LIN {X 0,Y 491.694,Z 547.992,A -85,B 0,C 180,E1 -6473.64,E2 -6473.64} C_VEL
LIN {X 0,Y 488.846,Z 539.593,A -85,B 0,C 180,E1 -6473.888,E2 -6473.888} C_VEL
LIN {X 0,Y 488.957,Z 539.577,A -85,B 0,C 180,E1 -6477.529,E2 -6477.529} C_VEL
LIN {X 0,Y 488.958,Z 539.578,A -85,B 0,C 180,E1 -6480,E2 -6480} C_VEL
LIN {X 0,Y 488.952,Z 539.582,A -85,B 0,C 180,E1 -6482.471,E2 -6482.471} C_VEL
LIN {X 0,Y 488.863,Z 539.586,A -85,B 0,C 180,E1 -6485.776,E2 -6485.776} C_VEL
LIN {X 0,Y 488.808,Z 539.594,A -85,B 0,C 180,E1 -6488.267,E2 -6488.267} C_VEL
LIN {X 0,Y 488.82,Z 539.592,A -85,B 0,C 180,E1 -6491.612,E2 -6491.612} C_VEL
LIN {X 0,Y 488.753,Z 539.602,A -85,B 0,C 180,E1 -6495.001,E2 -6495.001} C_VEL
LIN {X 0,Y 488.744,Z 539.606,A -85,B 0,C 180,E1 -6498.443,E2 -6498.443} C_VEL
LIN {X 0,Y 488.697,Z 539.611,A -85,B 0,C 180,E1 -6501.071,E2 -6501.071} C_VEL
LIN {X 0,Y 488.683,Z 539.609,A -85,B 0,C 180,E1 -6503.746,E2 -6503.746} C_VEL
LIN {X 0,Y 488.789,Z 539.601,A -85,B 0,C 180,E1 -6506.946,E2 -6506.946} C_VEL
LIN {X 0,Y 488.71,Z 539.608,A -85,B 0,C 180,E1 -6510.366,E2 -6510.366} C_VEL
LIN {X 0,Y 488.728,Z 539.604,A -85,B 0,C 180,E1 -6513.485,E2 -6513.485} C_VEL
LIN {X 0,Y 488.682,Z 539.612,A -85,B 0,C 180,E1 -6516.357,E2 -6516.357} C_VEL
LIN {X 0,Y 488.742,Z 539.604,A -85,B 0,C 180,E1 -6519.251,E2 -6519.251} C_VEL
LIN {X 0,Y 488.728,Z 539.609,A -85,B 0,C 180,E1 -6522.522,E2 -6522.522} C_VEL
LIN {X 0,Y 488.706,Z 539.611,A -85,B 0,C 180,E1 -6525.2,E2 -6525.2} C_VEL
LIN {X 0,Y 488.73,Z 539.605,A -85,B 0,C 180,E1 -6527.48,E2 -6527.48} C_VEL
LIN {X 0,Y 488.744,Z 539.607,A -85,B 0,C 180,E1 -6530.752,E2 -6530.752} C_VEL
LIN {X 0,Y 488.683,Z 539.612,A -85,B 0,C 180,E1 -6533.87,E2 -6533.87} C_VEL
LIN {X 0,Y 488.737,Z 539.61,A -85,B 0,C 180,E1 -6536.878,E2 -6536.878} C_VEL
LIN {X 0,Y 488.796,Z 539.749,A -85,B 0,C 180,E1 -6540.411,E2 -6540.411} C_VEL
LIN {X 0,Y 491.958,Z 554.443,A -85,B 0,C 180,E1 -6542.55,E2 -6542.55} C_VEL
LIN {X 0,Y 491.604,Z 568.227,A -85,B 0,C 180,E1 -6544.347,E2 -6544.347} C_VEL
LIN {X 0,Y 490.777,Z 592.773,A -85,B 0,C 180,E1 -6547.478,E2 -6547.478} C_VEL
LIN {X 0,Y 490.123,Z 615.461,A -85,B 0,C 180,E1 -6550.309,E2 -6550.309} C_VEL
LIN {X 0,Y 489.503,Z 641.425,A -85,B 0,C 180,E1 -6553.507,E2 -6553.507} C_VEL
LIN {X 0,Y 489.465,Z 643.124,A -85,B 0,C 180,E1 -6553.715,E2 -6553.715} C_VEL
LIN {X 0,Y 491.552,Z 663.555,A -85,B 0,C 180,E1 -6554.102,E2 -6554.102} C_VEL
LIN {X 0,Y 490.879,Z 754.427,A -85,B 0,C 180,E1 -6555.491,E2 -6555.491} C_VEL
LIN {X 0,Y 490.504,Z 768.429,A -85,B 0,C 180,E1 -6555.877,E2 -6555.877} C_VEL
LIN {X 0,Y 490.138,Z 781.627,A -85,B 0,C 180,E1 -6556.421,E2 -6556.421} C_VEL
LIN {X 0,Y 489.854,Z 793.54,A -85,B 0,C 180,E1 -6557.047,E2 -6557.047} C_VEL
LIN {X 0,Y 489.551,Z 804.345,A -85,B 0,C 180,E1 -6557.776,E2 -6557.776} C_VEL
LIN {X 0,Y 489.111,Z 815.314,A -85,B 0,C 180,E1 -6558.711,E2 -6558.711} C_VEL
LIN {X 0,Y 488.793,Z 824.213,A -85,B 0,C 180,E1 -6559.647,E2 -6559.647} C_VEL
LIN {X 0,Y 488.538,Z 832.373,A -85,B 0,C 180,E1 -6560.687,E2 -6560.687} C_VEL
LIN {X 0,Y 488.332,Z 840.353,A -85,B 0,C 180,E1 -6561.934,E2 -6561.934} C_VEL
LIN {X 0,Y 488.188,Z 845.733,A -85,B 0,C 180,E1 -6562.972,E2 -6562.972} C_VEL
LIN {X 0,Y 488.147,Z 850.985,A -85,B 0,C 180,E1 -6564.217,E2 -6564.217} C_VEL
LIN {X 0,Y 488.028,Z 855.04,A -85,B 0,C 180,E1 -6565.458,E2 -6565.458} C_VEL
LIN {X 0,Y 488.064,Z 858.028,A -85,B 0,C 180,E1 -6566.699,E2 -6566.699} C_VEL
LIN {X 0,Y 488.013,Z 859.461,A -85,B 0,C 180,E1 -6567.525,E2 -6567.525} C_VEL
LIN {X 0,Y 487.957,Z 861.087,A -85,B 0,C 180,E1 -6569.175,E2 -6569.175} C_VEL
LIN {X 0,Y 487.966,Z 861.309,A -85,B 0,C 180,E1 -6570.001,E2 -6570.001} C_VEL
LIN {X 0,Y 487.964,Z 860.468,A -85,B 0,C 180,E1 -6571.651,E2 -6571.651} C_VEL
LIN {X 0,Y 488.002,Z 859.457,A -85,B 0,C 180,E1 -6572.477,E2 -6572.477} C_VEL
LIN {X 0,Y 488.033,Z 858.023,A -85,B 0,C 180,E1 -6573.303,E2 -6573.303} C_VEL
LIN {X 0,Y 488.022,Z 855.034,A -85,B 0,C 180,E1 -6574.544,E2 -6574.544} C_VEL
LIN {X 0,Y 488.147,Z 849.944,A -85,B 0,C 180,E1 -6576.05,E2 -6576.05} C_VEL
LIN {X 0,Y 488.207,Z 843.696,A -85,B 0,C 180,E1 -6577.445,E2 -6577.445} C_VEL
LIN {X 0,Y 488.433,Z 836.567,A -85,B 0,C 180,E1 -6578.69,E2 -6578.69} C_VEL
LIN {X 0,Y 488.667,Z 827.667,A -85,B 0,C 180,E1 -6579.939,E2 -6579.939} C_VEL
LIN {X 0,Y 488.999,Z 818.502,A -85,B 0,C 180,E1 -6580.979,E2 -6580.979} C_VEL
LIN {X 0,Y 489.377,Z 808.262,A -85,B 0,C 180,E1 -6581.914,E2 -6581.914} C_VEL
LIN {X 0,Y 489.69,Z 797.091,A -85,B 0,C 180,E1 -6582.738,E2 -6582.738} C_VEL
LIN {X 0,Y 490.104,Z 784.736,A -85,B 0,C 180,E1 -6583.476,E2 -6583.476} C_VEL
LIN {X 0,Y 490.522,Z 771.929,A -85,B 0,C 180,E1 -6584.045,E2 -6584.045} C_VEL
LIN {X 0,Y 490.842,Z 759.389,A -85,B 0,C 180,E1 -6584.432,E2 -6584.432} C_VEL
LIN {X 0,Y 491.06,Z 742.038,A -85,B 0,C 180,E1 -6584.743,E2 -6584.743} C_VEL
LIN {X 0,Y 491.516,Z 663.042,A -85,B 0,C 180,E1 -6585.933,E2 -6585.933} C_VEL
LIN {X 0,Y 489.357,Z 645.546,A -85,B 0,C 180,E1 -6586.287,E2 -6586.287} C_VEL
LIN {X 0,Y 489.969,Z 622.617,A -85,B 0,C 180,E1 -6589.481,E2 -6589.481} C_VEL
LIN {X 0,Y 490.634,Z 601.006,A -85,B 0,C 180,E1 -6592.531,E2 -6592.531} C_VEL
LIN {X 0,Y 491.434,Z 579.535,A -85,B 0,C 180,E1 -6595.603,E2 -6595.603} C_VEL
LIN {X 0,Y 492.217,Z 559.133,A -85,B 0,C 180,E1 -6598.576,E2 -6598.576} C_VEL
LIN {X 0,Y 492.12,Z 554.913,A -85,B 0,C 180,E1 -6599.212,E2 -6599.212} C_VEL
LIN {X 0,Y 488.728,Z 539.608,A -85,B 0,C 180,E1 -6601.733,E2 -6601.733} C_VEL
LIN {X 0,Y 488.735,Z 539.604,A -85,B 0,C 180,E1 -6604.113,E2 -6604.113} C_VEL
LIN {X 0,Y 488.682,Z 539.616,A -85,B 0,C 180,E1 -6607.159,E2 -6607.159} C_VEL
LIN {X 0,Y 488.72,Z 539.605,A -85,B 0,C 180,E1 -6610.345,E2 -6610.345} C_VEL
LIN {X 0,Y 488.689,Z 539.604,A -85,B 0,C 180,E1 -6613.654,E2 -6613.654} C_VEL
LIN {X 0,Y 488.718,Z 539.604,A -85,B 0,C 180,E1 -6616.349,E2 -6616.349} C_VEL
LIN {X 0,Y 488.734,Z 539.604,A -85,B 0,C 180,E1 -6619.677,E2 -6619.677} C_VEL
LIN {X 0,Y 488.684,Z 539.61,A -85,B 0,C 180,E1 -6622.841,E2 -6622.841} C_VEL
LIN {X 0,Y 488.736,Z 539.603,A -85,B 0,C 180,E1 -6625.887,E2 -6625.887} C_VEL
LIN {X 0,Y 488.693,Z 539.605,A -85,B 0,C 180,E1 -6628.82,E2 -6628.82} C_VEL
LIN {X 0,Y 488.745,Z 539.604,A -85,B 0,C 180,E1 -6631.671,E2 -6631.671} C_VEL
LIN {X 0,Y 488.747,Z 539.595,A -85,B 0,C 180,E1 -6634.444,E2 -6634.444} C_VEL
LIN {X 0,Y 488.723,Z 539.604,A -85,B 0,C 180,E1 -6637.153,E2 -6637.153} C_VEL
LIN {X 0,Y 488.725,Z 539.604,A -85,B 0,C 180,E1 -6639.81,E2 -6639.81} C_VEL
LIN {X 0,Y 488.733,Z 539.592,A -85,B 0,C 180,E1 -6642.423,E2 -6642.423} C_VEL
LIN {X 0,Y 488.764,Z 539.599,A -85,B 0,C 180,E1 -6645,E2 -6645} C_VEL
LIN {X 0,Y 488.805,Z 539.587,A -85,B 0,C 180,E1 -6648.388,E2 -6648.388} C_VEL
LIN {X 0,Y 488.818,Z 539.597,A -85,B 0,C 180,E1 -6651.734,E2 -6651.734} C_VEL
LIN {X 0,Y 488.855,Z 539.587,A -85,B 0,C 180,E1 -6654.224,E2 -6654.224} C_VEL
LIN {X 0,Y 488.961,Z 539.57,A -85,B 0,C 180,E1 -6657.529,E2 -6657.529} C_VEL
LIN {X 0,Y 488.954,Z 539.574,A -85,B 0,C 180,E1 -6660.824,E2 -6660.824} C_VEL
LIN {X 0,Y 488.961,Z 539.572,A -85,B 0,C 180,E1 -6662.471,E2 -6662.471} C_VEL
LIN {X 0,Y 488.855,Z 539.584,A -85,B 0,C 180,E1 -6665.776,E2 -6665.776} C_VEL
LIN {X 0,Y 488.817,Z 539.594,A -85,B 0,C 180,E1 -6668.266,E2 -6668.266} C_VEL
LIN {X 0,Y 488.805,Z 539.594,A -85,B 0,C 180,E1 -6671.613,E2 -6671.613} C_VEL
LIN {X 0,Y 488.762,Z 539.597,A -85,B 0,C 180,E1 -6675,E2 -6675} C_VEL
LIN {X 0,Y 488.755,Z 539.594,A -85,B 0,C 180,E1 -6678.442,E2 -6678.442} C_VEL
LIN {X 0,Y 488.707,Z 539.603,A -85,B 0,C 180,E1 -6681.071,E2 -6681.071} C_VEL
LIN {X 0,Y 488.694,Z 539.612,A -85,B 0,C 180,E1 -6683.746,E2 -6683.746} C_VEL
LIN {X 0,Y 488.792,Z 539.593,A -85,B 0,C 180,E1 -6686.944,E2 -6686.944} C_VEL
LIN {X 0,Y 488.71,Z 539.605,A -85,B 0,C 180,E1 -6690.363,E2 -6690.363} C_VEL
LIN {X 0,Y 488.735,Z 539.604,A -85,B 0,C 180,E1 -6693.484,E2 -6693.484} C_VEL
LIN {X 0,Y 488.683,Z 539.615,A -85,B 0,C 180,E1 -6696.355,E2 -6696.355} C_VEL
LIN {X 0,Y 488.703,Z 539.605,A -85,B 0,C 180,E1 -6699.254,E2 -6699.254} C_VEL
LIN {X 0,Y 488.71,Z 539.607,A -85,B 0,C 180,E1 -6701.6,E2 -6701.6} C_VEL
LIN {X 0,Y 488.703,Z 539.608,A -85,B 0,C 180,E1 -6704.803,E2 -6704.803} C_VEL
LIN {X 0,Y 488.69,Z 539.598,A -85,B 0,C 180,E1 -6707.474,E2 -6707.474} C_VEL
LIN {X 0,Y 488.735,Z 539.604,A -85,B 0,C 180,E1 -6709.677,E2 -6709.677} C_VEL
LIN {X 0,Y 488.682,Z 539.612,A -85,B 0,C 180,E1 -6712.841,E2 -6712.841} C_VEL
LIN {X 0,Y 488.736,Z 539.606,A -85,B 0,C 180,E1 -6715.887,E2 -6715.887} C_VEL
LIN {X 0,Y 488.696,Z 539.616,A -85,B 0,C 180,E1 -6718.82,E2 -6718.82} C_VEL
LIN {X 0,Y 488.788,Z 539.603,A -85,B 0,C 180,E1 -6722.17,E2 -6722.17} C_VEL
LIN {X 0,Y 489.997,Z 545.204,A -85,B 0,C 180,E1 -6723.021,E2 -6723.021} C_VEL
LIN {X 0,Y 490.113,Z 548.909,A -85,B 0,C 180,E1 -6723.557,E2 -6723.557} C_VEL
LIN {X 0,Y 489.104,Z 552.826,A -85,B 0,C 180,E1 -6724.068,E2 -6724.068} C_VEL
LIN {X 0,Y 485.091,Z 563.467,A -85,B 0,C 180,E1 -6725.412,E2 -6725.412} C_VEL
LIN {X 0,Y 484.682,Z 566.068,A -85,B 0,C 180,E1 -6725.772,E2 -6725.772} C_VEL
LIN {X 0,Y 483.859,Z 586.48,A -85,B 0,C 180,E1 -6728.708,E2 -6728.708} C_VEL
LIN {X 0,Y 483.266,Z 606.74,A -85,B 0,C 180,E1 -6731.56,E2 -6731.56} C_VEL
LIN {X 0,Y 482.955,Z 621.519,A -85,B 0,C 180,E1 -6733.543,E2 -6733.543} C_VEL
LIN {X 0,Y 484.937,Z 634.789,A -85,B 0,C 180,E1 -6733.814,E2 -6733.814} C_VEL
LIN {X 0,Y 484.351,Z 730.687,A -85,B 0,C 180,E1 -6735.263,E2 -6735.263} C_VEL
LIN {X 0,Y 484.065,Z 743.533,A -85,B 0,C 180,E1 -6735.603,E2 -6735.603} C_VEL
LIN {X 0,Y 483.672,Z 756.506,A -85,B 0,C 180,E1 -6736.128,E2 -6736.128} C_VEL
LIN {X 0,Y 483.242,Z 769.444,A -85,B 0,C 180,E1 -6736.855,E2 -6736.855} C_VEL
LIN {X 0,Y 482.846,Z 781.021,A -85,B 0,C 180,E1 -6737.709,E2 -6737.709} C_VEL
LIN {X 0,Y 482.346,Z 792.291,A -85,B 0,C 180,E1 -6738.762,E2 -6738.762} C_VEL
LIN {X 0,Y 482.016,Z 800.524,A -85,B 0,C 180,E1 -6739.711,E2 -6739.711} C_VEL
LIN {X 0,Y 481.685,Z 808.123,A -85,B 0,C 180,E1 -6740.764,E2 -6740.764} C_VEL
LIN {X 0,Y 481.365,Z 815.544,A -85,B 0,C 180,E1 -6742.027,E2 -6742.027} C_VEL
LIN {X 0,Y 481.126,Z 821.834,A -85,B 0,C 180,E1 -6743.367,E2 -6743.367} C_VEL
LIN {X 0,Y 481.021,Z 826.219,A -85,B 0,C 180,E1 -6744.55,E2 -6744.55} C_VEL
LIN {X 0,Y 480.943,Z 829.827,A -85,B 0,C 180,E1 -6745.809,E2 -6745.809} C_VEL
LIN {X 0,Y 480.908,Z 831.685,A -85,B 0,C 180,E1 -6746.648,E2 -6746.648} C_VEL
LIN {X 0,Y 480.846,Z 833.109,A -85,B 0,C 180,E1 -6747.486,E2 -6747.486} C_VEL
LIN {X 0,Y 480.823,Z 834.106,A -85,B 0,C 180,E1 -6748.324,E2 -6748.324} C_VEL
LIN {X 0,Y 480.743,Z 834.962,A -85,B 0,C 180,E1 -6749.999,E2 -6749.999} C_VEL
LIN {X 0,Y 480.823,Z 834.192,A -85,B 0,C 180,E1 -6751.674,E2 -6751.674} C_VEL
LIN {X 0,Y 480.908,Z 831.872,A -85,B 0,C 180,E1 -6753.35,E2 -6753.35} C_VEL
LIN {X 0,Y 480.899,Z 829.015,A -85,B 0,C 180,E1 -6754.61,E2 -6754.61} C_VEL
LIN {X 0,Y 481.1,Z 825.127,A -85,B 0,C 180,E1 -6755.868,E2 -6755.868} C_VEL
LIN {X 0,Y 481.191,Z 820.1,A -85,B 0,C 180,E1 -6757.131,E2 -6757.131} C_VEL
LIN {X 0,Y 481.41,Z 813.759,A -85,B 0,C 180,E1 -6758.394,E2 -6758.394} C_VEL
LIN {X 0,Y 481.748,Z 805.871,A -85,B 0,C 180,E1 -6759.657,E2 -6759.657} C_VEL
LIN {X 0,Y 482.07,Z 797.812,A -85,B 0,C 180,E1 -6760.712,E2 -6760.712} C_VEL
LIN {X 0,Y 482.573,Z 787.935,A -85,B 0,C 180,E1 -6761.764,E2 -6761.764} C_VEL
LIN {X 0,Y 482.996,Z 776.744,A -85,B 0,C 180,E1 -6762.721,E2 -6762.721} C_VEL
LIN {X 0,Y 483.377,Z 766.004,A -85,B 0,C 180,E1 -6763.451,E2 -6763.451} C_VEL
LIN {X 0,Y 483.783,Z 753.895,A -85,B 0,C 180,E1 -6764.082,E2 -6764.082} C_VEL
LIN {X 0,Y 484.14,Z 740.567,A -85,B 0,C 180,E1 -6764.581,E2 -6764.581} C_VEL
LIN {X 0,Y 484.367,Z 727.094,A -85,B 0,C 180,E1 -6764.897,E2 -6764.897} C_VEL
LIN {X 0,Y 484.82,Z 635.15,A -85,B 0,C 180,E1 -6766.274,E2 -6766.274} C_VEL
LIN {X 0,Y 482.662,Z 622.172,A -85,B 0,C 180,E1 -6766.566,E2 -6766.566} C_VEL
LIN {X 0,Y 483.144,Z 602.516,A -85,B 0,C 180,E1 -6769.545,E2 -6769.545} C_VEL
LIN {X 0,Y 483.734,Z 584.445,A -85,B 0,C 180,E1 -6772.418,E2 -6772.418} C_VEL
LIN {X 0,Y 484.377,Z 566.321,A -85,B 0,C 180,E1 -6775.341,E2 -6775.341} C_VEL
LIN {X 0,Y 484.651,Z 554.986,A -85,B 0,C 180,E1 -6777.179,E2 -6777.179} C_VEL
LIN {X 0,Y 482.201,Z 542.669,A -85,B 0,C 180,E1 -6779.28,E2 -6779.28} C_VEL
LIN {X 0,Y 481.699,Z 540.486,A -85,B 0,C 180,E1 -6779.685,E2 -6779.685} C_VEL
LIN {X 0,Y 481.671,Z 540.486,A -85,B 0,C 180,E1 -6782.673,E2 -6782.673} C_VEL
LIN {X 0,Y 481.64,Z 540.488,A -85,B 0,C 180,E1 -6785.708,E2 -6785.708} C_VEL
LIN {X 0,Y 481.668,Z 540.488,A -85,B 0,C 180,E1 -6788.858,E2 -6788.858} C_VEL
LIN {X 0,Y 481.658,Z 540.484,A -85,B 0,C 180,E1 -6791.913,E2 -6791.913} C_VEL
LIN {X 0,Y 481.654,Z 540.48,A -85,B 0,C 180,E1 -6794.456,E2 -6794.456} C_VEL
LIN {X 0,Y 481.683,Z 540.483,A -85,B 0,C 180,E1 -6796.845,E2 -6796.845} C_VEL
LIN {X 0,Y 481.687,Z 540.483,A -85,B 0,C 180,E1 -6800.06,E2 -6800.06} C_VEL
LIN {X 0,Y 481.681,Z 540.499,A -85,B 0,C 180,E1 -6802.043,E2 -6802.043} C_VEL
LIN {X 0,Y 484.76,Z 549.63,A -85,B 0,C 180,E1 -6802.296,E2 -6802.296} C_VEL
LIN {X 0,Y 484.229,Z 619.899,A -85,B 0,C 180,E1 -6803.411,E2 -6803.411} C_VEL
LIN {X 0,Y 484.143,Z 632.566,A -85,B 0,C 180,E1 -6803.766,E2 -6803.766} C_VEL
LIN {X 0,Y 484.01,Z 645.447,A -85,B 0,C 180,E1 -6804.301,E2 -6804.301} C_VEL
LIN {X 0,Y 483.712,Z 657.474,A -85,B 0,C 180,E1 -6804.977,E2 -6804.977} C_VEL
LIN {X 0,Y 483.368,Z 668.816,A -85,B 0,C 180,E1 -6805.803,E2 -6805.803} C_VEL
LIN {X 0,Y 483.007,Z 679.79,A -85,B 0,C 180,E1 -6806.807,E2 -6806.807} C_VEL
LIN {X 0,Y 482.626,Z 689.455,A -85,B 0,C 180,E1 -6807.916,E2 -6807.916} C_VEL
LIN {X 0,Y 482.342,Z 697.942,A -85,B 0,C 180,E1 -6809.12,E2 -6809.12} C_VEL
LIN {X 0,Y 482.034,Z 704.631,A -85,B 0,C 180,E1 -6810.283,E2 -6810.283} C_VEL
LIN {X 0,Y 481.791,Z 711.107,A -85,B 0,C 180,E1 -6811.7,E2 -6811.7} C_VEL
LIN {X 0,Y 481.666,Z 715.997,A -85,B 0,C 180,E1 -6813.107,E2 -6813.107} C_VEL
LIN {X 0,Y 481.58,Z 718.529,A -85,B 0,C 180,E1 -6814.036,E2 -6814.036} C_VEL
LIN {X 0,Y 481.487,Z 720.459,A -85,B 0,C 180,E1 -6814.957,E2 -6814.957} C_VEL
LIN {X 0,Y 481.429,Z 721.907,A -85,B 0,C 180,E1 -6815.874,E2 -6815.874} C_VEL
LIN {X 0,Y 481.389,Z 722.929,A -85,B 0,C 180,E1 -6816.888,E2 -6816.888} C_VEL
LIN {X 0,Y 481.405,Z 723.32,A -85,B 0,C 180,E1 -6817.693,E2 -6817.693} C_VEL
LIN {X 0,Y 481.417,Z 723.133,A -85,B 0,C 180,E1 -6819.112,E2 -6819.112} C_VEL
LIN {X 0,Y 481.477,Z 721.986,A -85,B 0,C 180,E1 -6820.383,E2 -6820.383} C_VEL
LIN {X 0,Y 481.598,Z 720.132,A -85,B 0,C 180,E1 -6821.536,E2 -6821.536} C_VEL
LIN {X 0,Y 481.746,Z 716.495,A -85,B 0,C 180,E1 -6823.036,E2 -6823.036} C_VEL
LIN {X 0,Y 481.951,Z 711.888,A -85,B 0,C 180,E1 -6824.4,E2 -6824.4} C_VEL
LIN {X 0,Y 482.242,Z 705.298,A -85,B 0,C 180,E1 -6825.871,E2 -6825.871} C_VEL
LIN {X 0,Y 482.564,Z 697.739,A -85,B 0,C 180,E1 -6827.189,E2 -6827.189} C_VEL
LIN {X 0,Y 482.835,Z 690.295,A -85,B 0,C 180,E1 -6828.242,E2 -6828.242} C_VEL
LIN {X 0,Y 483.213,Z 681.009,A -85,B 0,C 180,E1 -6829.313,E2 -6829.313} C_VEL
LIN {X 0,Y 483.592,Z 670.655,A -85,B 0,C 180,E1 -6830.273,E2 -6830.273} C_VEL
LIN {X 0,Y 483.918,Z 659.298,A -85,B 0,C 180,E1 -6831.115,E2 -6831.115} C_VEL
LIN {X 0,Y 484.181,Z 646.995,A -85,B 0,C 180,E1 -6831.811,E2 -6831.811} C_VEL
LIN {X 0,Y 484.306,Z 633.622,A -85,B 0,C 180,E1 -6832.364,E2 -6832.364} C_VEL
LIN {X 0,Y 484.364,Z 620.986,A -85,B 0,C 180,E1 -6832.706,E2 -6832.706} C_VEL
LIN {X 0,Y 484.864,Z 549.455,A -85,B 0,C 180,E1 -6833.863,E2 -6833.863} C_VEL
LIN {X 0,Y 481.827,Z 540.469,A -85,B 0,C 180,E1 -6834.14,E2 -6834.14} C_VEL
LIN {X 0,Y 481.924,Z 540.453,A -85,B 0,C 180,E1 -6837.492,E2 -6837.492} C_VEL
LIN {X 0,Y 481.929,Z 540.454,A -85,B 0,C 180,E1 -6840,E2 -6840} C_VEL
LIN {X 0,Y 481.919,Z 540.458,A -85,B 0,C 180,E1 -6842.507,E2 -6842.507} C_VEL
LIN {X 0,Y 481.821,Z 540.464,A -85,B 0,C 180,E1 -6845.86,E2 -6845.86} C_VEL
LIN {X 0,Y 481.753,Z 540.474,A -85,B 0,C 180,E1 -6848.388,E2 -6848.388} C_VEL
LIN {X 0,Y 481.784,Z 540.469,A -85,B 0,C 180,E1 -6851.784,E2 -6851.784} C_VEL
LIN {X 0,Y 481.733,Z 540.473,A -85,B 0,C 180,E1 -6855.225,E2 -6855.225} C_VEL
LIN {X 0,Y 481.702,Z 540.485,A -85,B 0,C 180,E1 -6858.722,E2 -6858.722} C_VEL
LIN {X 0,Y 481.637,Z 540.488,A -85,B 0,C 180,E1 -6861.395,E2 -6861.395} C_VEL
LIN {X 0,Y 481.667,Z 540.484,A -85,B 0,C 180,E1 -6864.114,E2 -6864.114} C_VEL
LIN {X 0,Y 481.742,Z 540.476,A -85,B 0,C 180,E1 -6867.141,E2 -6867.141} C_VEL
LIN {X 0,Y 481.679,Z 540.481,A -85,B 0,C 180,E1 -6869.741,E2 -6869.741} C_VEL
LIN {X 0,Y 481.665,Z 540.489,A -85,B 0,C 180,E1 -6872.675,E2 -6872.675} C_VEL
LIN {X 0,Y 481.636,Z 540.487,A -85,B 0,C 180,E1 -6875.71,E2 -6875.71} C_VEL
LIN {X 0,Y 481.713,Z 540.479,A -85,B 0,C 180,E1 -6879.356,E2 -6879.356} C_VEL
LIN {X 0,Y 481.669,Z 540.485,A -85,B 0,C 180,E1 -6882.159,E2 -6882.159} C_VEL
LIN {X 0,Y 481.654,Z 540.49,A -85,B 0,C 180,E1 -6884.458,E2 -6884.458} C_VEL
LIN {X 0,Y 481.684,Z 540.487,A -85,B 0,C 180,E1 -6886.847,E2 -6886.847} C_VEL
LIN {X 0,Y 481.688,Z 540.482,A -85,B 0,C 180,E1 -6890.062,E2 -6890.062} C_VEL
LIN {X 0,Y 481.628,Z 540.494,A -85,B 0,C 180,E1 -6893.255,E2 -6893.255} C_VEL
LIN {X 0,Y 481.706,Z 540.482,A -85,B 0,C 180,E1 -6896.331,E2 -6896.331} C_VEL
LIN {X 0,Y 481.69,Z 540.486,A -85,B 0,C 180,E1 -6899.778,E2 -6899.778} C_VEL
LIN {X 0,Y 481.682,Z 540.506,A -85,B 0,C 180,E1 -6900.14,E2 -6900.14} C_VEL
LIN {X 0,Y 484.991,Z 555.483,A -85,B 0,C 180,E1 -6902.374,E2 -6902.374} C_VEL
LIN {X 0,Y 484.898,Z 563.926,A -85,B 0,C 180,E1 -6903.51,E2 -6903.51} C_VEL
LIN {X 0,Y 484.044,Z 586.865,A -85,B 0,C 180,E1 -6906.502,E2 -6906.502} C_VEL
LIN {X 0,Y 483.295,Z 609.138,A -85,B 0,C 180,E1 -6909.352,E2 -6909.352} C_VEL
LIN {X 0,Y 482.634,Z 633.496,A -85,B 0,C 180,E1 -6912.414,E2 -6912.414} C_VEL
LIN {X 0,Y 482.43,Z 641.831,A -85,B 0,C 180,E1 -6913.454,E2 -6913.454} C_VEL
LIN {X 0,Y 484.679,Z 663.774,A -85,B 0,C 180,E1 -6913.893,E2 -6913.893} C_VEL
LIN {X 0,Y 483.941,Z 753.875,A -85,B 0,C 180,E1 -6915.305,E2 -6915.305} C_VEL
LIN {X 0,Y 483.538,Z 767.693,A -85,B 0,C 180,E1 -6915.696,E2 -6915.696} C_VEL
LIN {X 0,Y 483.233,Z 781.439,A -85,B 0,C 180,E1 -6916.223,E2 -6916.223} C_VEL
LIN {X 0,Y 482.906,Z 793.909,A -85,B 0,C 180,E1 -6916.889,E2 -6916.889} C_VEL
LIN {X 0,Y 482.515,Z 805.432,A -85,B 0,C 180,E1 -6917.694,E2 -6917.694} C_VEL
LIN {X 0,Y 482.09,Z 816.209,A -85,B 0,C 180,E1 -6918.651,E2 -6918.651} C_VEL
LIN {X 0,Y 481.713,Z 825.818,A -85,B 0,C 180,E1 -6919.706,E2 -6919.706} C_VEL
LIN {X 0,Y 481.439,Z 833.672,A -85,B 0,C 180,E1 -6920.76,E2 -6920.76} C_VEL
LIN {X 0,Y 481.23,Z 841.303,A -85,B 0,C 180,E1 -6922.026,E2 -6922.026} C_VEL
LIN {X 0,Y 481.028,Z 848.192,A -85,B 0,C 180,E1 -6923.468,E2 -6923.468} C_VEL
LIN {X 0,Y 481.023,Z 852.248,A -85,B 0,C 180,E1 -6924.551,E2 -6924.551} C_VEL
LIN {X 0,Y 480.97,Z 855.936,A -85,B 0,C 180,E1 -6925.811,E2 -6925.811} C_VEL
LIN {X 0,Y 480.986,Z 857.836,A -85,B 0,C 180,E1 -6926.65,E2 -6926.65} C_VEL
LIN {X 0,Y 480.922,Z 859.268,A -85,B 0,C 180,E1 -6927.488,E2 -6927.488} C_VEL
LIN {X 0,Y 480.897,Z 860.278,A -85,B 0,C 180,E1 -6928.326,E2 -6928.326} C_VEL
LIN {X 0,Y 480.875,Z 860.895,A -85,B 0,C 180,E1 -6929.163,E2 -6929.163} C_VEL
LIN {X 0,Y 480.881,Z 861.116,A -85,B 0,C 180,E1 -6930.001,E2 -6930.001} C_VEL
LIN {X 0,Y 480.891,Z 860.276,A -85,B 0,C 180,E1 -6931.676,E2 -6931.676} C_VEL
LIN {X 0,Y 480.911,Z 859.265,A -85,B 0,C 180,E1 -6932.513,E2 -6932.513} C_VEL
LIN {X 0,Y 480.958,Z 857.831,A -85,B 0,C 180,E1 -6933.351,E2 -6933.351} C_VEL
LIN {X 0,Y 480.931,Z 854.843,A -85,B 0,C 180,E1 -6934.611,E2 -6934.611} C_VEL
LIN {X 0,Y 481.047,Z 850.789,A -85,B 0,C 180,E1 -6935.87,E2 -6935.87} C_VEL
LIN {X 0,Y 481.116,Z 844.521,A -85,B 0,C 180,E1 -6937.344,E2 -6937.344} C_VEL
LIN {X 0,Y 481.329,Z 837.682,A -85,B 0,C 180,E1 -6938.608,E2 -6938.608} C_VEL
LIN {X 0,Y 481.532,Z 830.689,A -85,B 0,C 180,E1 -6939.663,E2 -6939.663} C_VEL
LIN {X 0,Y 481.801,Z 822.23,A -85,B 0,C 180,E1 -6940.719,E2 -6940.719} C_VEL
LIN {X 0,Y 482.209,Z 811.732,A -85,B 0,C 180,E1 -6941.774,E2 -6941.774} C_VEL
LIN {X 0,Y 482.535,Z 801.308,A -85,B 0,C 180,E1 -6942.62,E2 -6942.62} C_VEL
LIN {X 0,Y 482.982,Z 789.785,A -85,B 0,C 180,E1 -6943.357,E2 -6943.357} C_VEL
LIN {X 0,Y 483.485,Z 774.679,A -85,B 0,C 180,E1 -6944.093,E2 -6944.093} C_VEL
LIN {X 0,Y 483.852,Z 761.919,A -85,B 0,C 180,E1 -6944.538,E2 -6944.538} C_VEL
LIN {X 0,Y 484.123,Z 748.987,A -85,B 0,C 180,E1 -6944.825,E2 -6944.825} C_VEL
LIN {X 0,Y 484.641,Z 663.611,A -85,B 0,C 180,E1 -6946.143,E2 -6946.143} C_VEL
LIN {X 0,Y 482.358,Z 644.648,A -85,B 0,C 180,E1 -6946.534,E2 -6946.534} C_VEL
LIN {X 0,Y 483.014,Z 621.8,A -85,B 0,C 180,E1 -6949.773,E2 -6949.773} C_VEL
LIN {X 0,Y 483.71,Z 600.186,A -85,B 0,C 180,E1 -6952.872,E2 -6952.872} C_VEL
LIN {X 0,Y 484.565,Z 578.409,A -85,B 0,C 180,E1 -6956.042,E2 -6956.042} C_VEL
LIN {X 0,Y 485.377,Z 558.339,A -85,B 0,C 180,E1 -6959.017,E2 -6959.017} C_VEL
LIN {X 0,Y 484.249,Z 551.933,A -85,B 0,C 180,E1 -6960.046,E2 -6960.046} C_VEL
LIN {X 0,Y 481.663,Z 540.488,A -85,B 0,C 180,E1 -6962,E2 -6962} C_VEL
LIN {X 0,Y 481.693,Z 540.485,A -85,B 0,C 180,E1 -6964.682,E2 -6964.682} C_VEL
LIN {X 0,Y 481.657,Z 540.484,A -85,B 0,C 180,E1 -6968.007,E2 -6968.007} C_VEL
LIN {X 0,Y 481.658,Z 540.491,A -85,B 0,C 180,E1 -6971.042,E2 -6971.042} C_VEL
LIN {X 0,Y 481.661,Z 540.479,A -85,B 0,C 180,E1 -6974.457,E2 -6974.457} C_VEL
LIN {X 0,Y 481.685,Z 540.485,A -85,B 0,C 180,E1 -6976.846,E2 -6976.846} C_VEL
LIN {X 0,Y 481.678,Z 540.481,A -85,B 0,C 180,E1 -6980.06,E2 -6980.06} C_VEL
LIN {X 0,Y 481.63,Z 540.487,A -85,B 0,C 180,E1 -6983.253,E2 -6983.253} C_VEL
LIN {X 0,Y 481.71,Z 540.477,A -85,B 0,C 180,E1 -6986.33,E2 -6986.33} C_VEL
LIN {X 0,Y 481.651,Z 540.484,A -85,B 0,C 180,E1 -6989.417,E2 -6989.417} C_VEL
LIN {X 0,Y 481.7,Z 540.478,A -85,B 0,C 180,E1 -6992.168,E2 -6992.168} C_VEL
LIN {X 0,Y 481.717,Z 540.474,A -85,B 0,C 180,E1 -6994.97,E2 -6994.97} C_VEL
LIN {X 0,Y 481.649,Z 540.489,A -85,B 0,C 180,E1 -6997.705,E2 -6997.705} C_VEL
LIN {X 0,Y 481.705,Z 540.474,A -85,B 0,C 180,E1 -7000.393,E2 -7000.393} C_VEL
LIN {X 0,Y 481.691,Z 540.472,A -85,B 0,C 180,E1 -7003.034,E2 -7003.034} C_VEL
LIN {X 0,Y 481.694,Z 540.485,A -85,B 0,C 180,E1 -7005.639,E2 -7005.639} C_VEL
LIN {X 0,Y 481.75,Z 540.466,A -85,B 0,C 180,E1 -7008.215,E2 -7008.215} C_VEL
LIN {X 0,Y 481.763,Z 540.473,A -85,B 0,C 180,E1 -7011.612,E2 -7011.612} C_VEL
LIN {X 0,Y 481.816,Z 540.464,A -85,B 0,C 180,E1 -7014.14,E2 -7014.14} C_VEL
LIN {X 0,Y 481.927,Z 540.445,A -85,B 0,C 180,E1 -7017.493,E2 -7017.493} C_VEL
LIN {X 0,Y 481.905,Z 540.452,A -85,B 0,C 180,E1 -7020.836,E2 -7020.836} C_VEL
LIN {X 0,Y 481.928,Z 540.448,A -85,B 0,C 180,E1 -7022.508,E2 -7022.508} C_VEL
LIN {X 0,Y 481.816,Z 540.462,A -85,B 0,C 180,E1 -7025.86,E2 -7025.86} C_VEL
LIN {X 0,Y 481.763,Z 540.472,A -85,B 0,C 180,E1 -7028.388,E2 -7028.388} C_VEL
LIN {X 0,Y 481.75,Z 540.47,A -85,B 0,C 180,E1 -7031.785,E2 -7031.785} C_VEL
LIN {X 0,Y 481.742,Z 540.473,A -85,B 0,C 180,E1 -7035.224,E2 -7035.224} C_VEL
LIN {X 0,Y 481.712,Z 540.469,A -85,B 0,C 180,E1 -7038.722,E2 -7038.722} C_VEL
LIN {X 0,Y 481.646,Z 540.484,A -85,B 0,C 180,E1 -7041.395,E2 -7041.395} C_VEL
LIN {X 0,Y 481.678,Z 540.482,A -85,B 0,C 180,E1 -7044.113,E2 -7044.113} C_VEL
LIN {X 0,Y 481.747,Z 540.471,A -85,B 0,C 180,E1 -7047.139,E2 -7047.139} C_VEL
LIN {X 0,Y 481.679,Z 540.484,A -85,B 0,C 180,E1 -7049.741,E2 -7049.741} C_VEL
LIN {X 0,Y 481.672,Z 540.484,A -85,B 0,C 180,E1 -7052.674,E2 -7052.674} C_VEL
LIN {X 0,Y 481.637,Z 540.486,A -85,B 0,C 180,E1 -7055.71,E2 -7055.71} C_VEL
LIN {X 0,Y 481.672,Z 540.481,A -85,B 0,C 180,E1 -7058.859,E2 -7058.859} C_VEL
LIN {X 0,Y 481.655,Z 540.49,A -85,B 0,C 180,E1 -7061.913,E2 -7061.913} C_VEL
LIN {X 0,Y 481.657,Z 540.489,A -85,B 0,C 180,E1 -7064.458,E2 -7064.458} C_VEL
LIN {X 0,Y 481.648,Z 540.477,A -85,B 0,C 180,E1 -7067.839,E2 -7067.839} C_VEL
LIN {X 0,Y 481.682,Z 540.482,A -85,B 0,C 180,E1 -7070.651,E2 -7070.651} C_VEL
LIN {X 0,Y 481.631,Z 540.488,A -85,B 0,C 180,E1 -7073.376,E2 -7073.376} C_VEL
LIN {X 0,Y 481.713,Z 540.484,A -85,B 0,C 180,E1 -7076.33,E2 -7076.33} C_VEL
LIN {X 0,Y 481.654,Z 540.49,A -85,B 0,C 180,E1 -7079.417,E2 -7079.417} C_VEL
LIN {X 0,Y 481.738,Z 540.673,A -85,B 0,C 180,E1 -7081.963,E2 -7081.963} C_VEL
LIN {X 0,Y 484.878,Z 555.303,A -85,B 0,C 180,E1 -7084.225,E2 -7084.225} C_VEL
LIN {X 0,Y 484.682,Z 566.068,A -85,B 0,C 180,E1 -7085.772,E2 -7085.772} C_VEL
LIN {X 0,Y 483.831,Z 569.916,A -85,B 0,C 180,E1 -7086.294,E2 -7086.294} C_VEL
LIN {X 0,Y 477.705,Z 582.954,A -85,B 0,C 180,E1 -7087.927,E2 -7087.927} C_VEL
LIN {X 0,Y 476.962,Z 586.803,A -85,B 0,C 180,E1 -7088.46,E2 -7088.46} C_VEL
LIN {X 0,Y 476.346,Z 606.679,A -85,B 0,C 180,E1 -7091.282,E2 -7091.282} C_VEL
LIN {X 0,Y 476.055,Z 621.776,A -85,B 0,C 180,E1 -7093.3,E2 -7093.3} C_VEL
LIN {X 0,Y 478.157,Z 636.429,A -85,B 0,C 180,E1 -7093.602,E2 -7093.602} C_VEL
LIN {X 0,Y 477.455,Z 732.033,A -85,B 0,C 180,E1 -7095.072,E2 -7095.072} C_VEL
LIN {X 0,Y 477.154,Z 745.254,A -85,B 0,C 180,E1 -7095.444,E2 -7095.444} C_VEL
LIN {X 0,Y 476.751,Z 757.717,A -85,B 0,C 180,E1 -7095.976,E2 -7095.976} C_VEL
LIN {X 0,Y 476.322,Z 769.933,A -85,B 0,C 180,E1 -7096.681,E2 -7096.681} C_VEL
LIN {X 0,Y 475.926,Z 781.195,A -85,B 0,C 180,E1 -7097.527,E2 -7097.527} C_VEL
LIN {X 0,Y 475.373,Z 792.472,A -85,B 0,C 180,E1 -7098.595,E2 -7098.595} C_VEL
LIN {X 0,Y 475.035,Z 800.708,A -85,B 0,C 180,E1 -7099.558,E2 -7099.558} C_VEL
LIN {X 0,Y 474.658,Z 808.311,A -85,B 0,C 180,E1 -7100.626,E2 -7100.626} C_VEL
LIN {X 0,Y 474.319,Z 815.733,A -85,B 0,C 180,E1 -7101.907,E2 -7101.907} C_VEL
LIN {X 0,Y 474.075,Z 822.332,A -85,B 0,C 180,E1 -7103.343,E2 -7103.343} C_VEL
LIN {X 0,Y 473.971,Z 826.411,A -85,B 0,C 180,E1 -7104.469,E2 -7104.469} C_VEL
LIN {X 0,Y 473.845,Z 830.02,A -85,B 0,C 180,E1 -7105.746,E2 -7105.746} C_VEL
LIN {X 0,Y 473.838,Z 831.878,A -85,B 0,C 180,E1 -7106.598,E2 -7106.598} C_VEL
LIN {X 0,Y 473.763,Z 833.302,A -85,B 0,C 180,E1 -7107.449,E2 -7107.449} C_VEL
LIN {X 0,Y 473.689,Z 834.916,A -85,B 0,C 180,E1 -7109.149,E2 -7109.149} C_VEL
LIN {X 0,Y 473.67,Z 835.154,A -85,B 0,C 180,E1 -7109.999,E2 -7109.999} C_VEL
LIN {X 0,Y 473.689,Z 834.967,A -85,B 0,C 180,E1 -7110.849,E2 -7110.849} C_VEL
LIN {X 0,Y 473.763,Z 833.421,A -85,B 0,C 180,E1 -7112.55,E2 -7112.55} C_VEL
LIN {X 0,Y 473.838,Z 832.062,A -85,B 0,C 180,E1 -7113.4,E2 -7113.4} C_VEL
LIN {X 0,Y 473.812,Z 829.205,A -85,B 0,C 180,E1 -7114.679,E2 -7114.679} C_VEL
LIN {X 0,Y 474.041,Z 825.314,A -85,B 0,C 180,E1 -7115.956,E2 -7115.956} C_VEL
LIN {X 0,Y 474.141,Z 820.285,A -85,B 0,C 180,E1 -7117.237,E2 -7117.237} C_VEL
LIN {X 0,Y 474.384,Z 813.941,A -85,B 0,C 180,E1 -7118.519,E2 -7118.519} C_VEL
LIN {X 0,Y 474.724,Z 806.048,A -85,B 0,C 180,E1 -7119.801,E2 -7119.801} C_VEL
LIN {X 0,Y 475.07,Z 797.984,A -85,B 0,C 180,E1 -7120.871,E2 -7120.871} C_VEL
LIN {X 0,Y 475.633,Z 788.099,A -85,B 0,C 180,E1 -7121.938,E2 -7121.938} C_VEL
LIN {X 0,Y 476.075,Z 776.777,A -85,B 0,C 180,E1 -7122.918,E2 -7122.918} C_VEL
LIN {X 0,Y 476.471,Z 766.147,A -85,B 0,C 180,E1 -7123.65,E2 -7123.65} C_VEL
LIN {X 0,Y 476.925,Z 754.012,A -85,B 0,C 180,E1 -7124.289,E2 -7124.289} C_VEL
LIN {X 0,Y 477.286,Z 740.647,A -85,B 0,C 180,E1 -7124.795,E2 -7124.795} C_VEL
LIN {X 0,Y 477.463,Z 728.619,A -85,B 0,C 180,E1 -7125.09,E2 -7125.09} C_VEL
LIN {X 0,Y 478.133,Z 636.899,A -85,B 0,C 180,E1 -7126.482,E2 -7126.482} C_VEL
LIN {X 0,Y 475.721,Z 622.347,A -85,B 0,C 180,E1 -7126.799,E2 -7126.799} C_VEL
LIN {X 0,Y 476.202,Z 603.746,A -85,B 0,C 180,E1 -7129.628,E2 -7129.628} C_VEL
LIN {X 0,Y 476.812,Z 585.626,A -85,B 0,C 180,E1 -7132.533,E2 -7132.533} C_VEL
LIN {X 0,Y 477.5,Z 567.395,A -85,B 0,C 180,E1 -7135.499,E2 -7135.499} C_VEL
LIN {X 0,Y 477.738,Z 556.188,A -85,B 0,C 180,E1 -7137.334,E2 -7137.334} C_VEL
LIN {X 0,Y 475.281,Z 544.116,A -85,B 0,C 180,E1 -7139.424,E2 -7139.424} C_VEL
LIN {X 0,Y 474.639,Z 541.365,A -85,B 0,C 180,E1 -7139.92,E2 -7139.92} C_VEL
LIN {X 0,Y 474.64,Z 541.362,A -85,B 0,C 180,E1 -7143.219,E2 -7143.219} C_VEL
LIN {X 0,Y 474.591,Z 541.364,A -85,B 0,C 180,E1 -7146.322,E2 -7146.322} C_VEL
LIN {X 0,Y 474.623,Z 541.361,A -85,B 0,C 180,E1 -7149.647,E2 -7149.647} C_VEL
LIN {X 0,Y 474.635,Z 541.359,A -85,B 0,C 180,E1 -7152.93,E2 -7152.93} C_VEL
LIN {X 0,Y 474.613,Z 541.363,A -85,B 0,C 180,E1 -7155.895,E2 -7155.895} C_VEL
LIN {X 0,Y 474.64,Z 541.363,A -85,B 0,C 180,E1 -7159.037,E2 -7159.037} C_VEL
LIN {X 0,Y 474.682,Z 541.534,A -85,B 0,C 180,E1 -7161.819,E2 -7161.819} C_VEL
LIN {X 0,Y 477.972,Z 551.217,A -85,B 0,C 180,E1 -7162.093,E2 -7162.093} C_VEL
LIN {X 0,Y 477.367,Z 620.718,A -85,B 0,C 180,E1 -7163.217,E2 -7163.217} C_VEL
LIN {X 0,Y 477.27,Z 633.206,A -85,B 0,C 180,E1 -7163.569,E2 -7163.569} C_VEL
LIN {X 0,Y 477.137,Z 646.032,A -85,B 0,C 180,E1 -7164.106,E2 -7164.106} C_VEL
LIN {X 0,Y 476.843,Z 658.117,A -85,B 0,C 180,E1 -7164.788,E2 -7164.788} C_VEL
LIN {X 0,Y 476.48,Z 669.361,A -85,B 0,C 180,E1 -7165.613,E2 -7165.613} C_VEL
LIN {X 0,Y 476.083,Z 680.522,A -85,B 0,C 180,E1 -7166.64,E2 -7166.64} C_VEL
LIN {X 0,Y 475.715,Z 689.707,A -85,B 0,C 180,E1 -7167.694,E2 -7167.694} C_VEL
LIN {X 0,Y 475.407,Z 697.858,A -85,B 0,C 180,E1 -7168.841,E2 -7168.841} C_VEL
LIN {X 0,Y 475.095,Z 704.881,A -85,B 0,C 180,E1 -7170.049,E2 -7170.049} C_VEL
LIN {X 0,Y 474.881,Z 710.63,A -85,B 0,C 180,E1 -7171.269,E2 -7171.269} C_VEL
LIN {X 0,Y 474.705,Z 715.872,A -85,B 0,C 180,E1 -7172.68,E2 -7172.68} C_VEL
LIN {X 0,Y 474.548,Z 719.764,A -85,B 0,C 180,E1 -7174.094,E2 -7174.094} C_VEL
LIN {X 0,Y 474.437,Z 722.411,A -85,B 0,C 180,E1 -7175.495,E2 -7175.495} C_VEL
LIN {X 0,Y 474.376,Z 723.827,A -85,B 0,C 180,E1 -7176.71,E2 -7176.71} C_VEL
LIN {X 0,Y 474.385,Z 724.4,A -85,B 0,C 180,E1 -7178.261,E2 -7178.261} C_VEL
LIN {X 0,Y 474.406,Z 724.133,A -85,B 0,C 180,E1 -7179.173,E2 -7179.173} C_VEL
LIN {X 0,Y 474.441,Z 723.432,A -85,B 0,C 180,E1 -7180.08,E2 -7180.08} C_VEL
LIN {X 0,Y 474.565,Z 721.547,A -85,B 0,C 180,E1 -7181.4,E2 -7181.4} C_VEL
LIN {X 0,Y 474.728,Z 718.476,A -85,B 0,C 180,E1 -7182.777,E2 -7182.777} C_VEL
LIN {X 0,Y 474.921,Z 714.298,A -85,B 0,C 180,E1 -7184.125,E2 -7184.125} C_VEL
LIN {X 0,Y 475.199,Z 707.986,A -85,B 0,C 180,E1 -7185.657,E2 -7185.657} C_VEL
LIN {X 0,Y 475.555,Z 700.956,A -85,B 0,C 180,E1 -7186.975,E2 -7186.975} C_VEL
LIN {X 0,Y 475.909,Z 692.149,A -85,B 0,C 180,E1 -7188.284,E2 -7188.284} C_VEL
LIN {X 0,Y 476.304,Z 683.07,A -85,B 0,C 180,E1 -7189.371,E2 -7189.371} C_VEL
LIN {X 0,Y 476.678,Z 672.966,A -85,B 0,C 180,E1 -7190.345,E2 -7190.345} C_VEL
LIN {X 0,Y 477.049,Z 661.54,A -85,B 0,C 180,E1 -7191.222,E2 -7191.222} C_VEL
LIN {X 0,Y 477.368,Z 650.081,A -85,B 0,C 180,E1 -7191.907,E2 -7191.907} C_VEL
LIN {X 0,Y 477.497,Z 638.182,A -85,B 0,C 180,E1 -7192.441,E2 -7192.441} C_VEL
LIN {X 0,Y 477.538,Z 625.329,A -85,B 0,C 180,E1 -7192.84,E2 -7192.84} C_VEL
LIN {X 0,Y 477.673,Z 599.465,A -85,B 0,C 180,E1 -7193.293,E2 -7193.293} C_VEL
LIN {X 0,Y 478.1,Z 550.884,A -85,B 0,C 180,E1 -7194.094,E2 -7194.094} C_VEL
LIN {X 0,Y 474.778,Z 541.349,A -85,B 0,C 180,E1 -7194.399,E2 -7194.399} C_VEL
LIN {X 0,Y 474.891,Z 541.329,A -85,B 0,C 180,E1 -7197.455,E2 -7197.455} C_VEL
LIN {X 0,Y 474.867,Z 541.338,A -85,B 0,C 180,E1 -7200.848,E2 -7200.848} C_VEL
LIN {X 0,Y 474.885,Z 541.335,A -85,B 0,C 180,E1 -7202.545,E2 -7202.545} C_VEL
LIN {X 0,Y 474.781,Z 541.341,A -85,B 0,C 180,E1 -7205.948,E2 -7205.948} C_VEL
LIN {X 0,Y 474.718,Z 541.352,A -85,B 0,C 180,E1 -7208.514,E2 -7208.514} C_VEL
LIN {X 0,Y 474.728,Z 541.348,A -85,B 0,C 180,E1 -7211.962,E2 -7211.962} C_VEL
LIN {X 0,Y 474.67,Z 541.351,A -85,B 0,C 180,E1 -7215.768,E2 -7215.768} C_VEL
LIN {X 0,Y 474.655,Z 541.361,A -85,B 0,C 180,E1 -7219.011,E2 -7219.011} C_VEL
LIN {X 0,Y 474.579,Z 541.366,A -85,B 0,C 180,E1 -7221.729,E2 -7221.729} C_VEL
LIN {X 0,Y 474.649,Z 541.362,A -85,B 0,C 180,E1 -7224.493,E2 -7224.493} C_VEL
LIN {X 0,Y 474.689,Z 541.353,A -85,B 0,C 180,E1 -7227.339,E2 -7227.339} C_VEL
LIN {X 0,Y 474.601,Z 541.369,A -85,B 0,C 180,E1 -7230.812,E2 -7230.812} C_VEL
LIN {X 0,Y 474.63,Z 541.359,A -85,B 0,C 180,E1 -7233.985,E2 -7233.985} C_VEL
LIN {X 0,Y 474.569,Z 541.371,A -85,B 0,C 180,E1 -7236.901,E2 -7236.901} C_VEL
LIN {X 0,Y 474.648,Z 541.357,A -85,B 0,C 180,E1 -7239.653,E2 -7239.653} C_VEL
LIN {X 0,Y 474.646,Z 541.363,A -85,B 0,C 180,E1 -7242.931,E2 -7242.931} C_VEL
LIN {X 0,Y 474.612,Z 541.363,A -85,B 0,C 180,E1 -7245.897,E2 -7245.897} C_VEL
LIN {X 0,Y 474.64,Z 541.363,A -85,B 0,C 180,E1 -7249.039,E2 -7249.039} C_VEL
LIN {X 0,Y 474.616,Z 541.363,A -85,B 0,C 180,E1 -7251.703,E2 -7251.703} C_VEL
LIN {X 0,Y 474.627,Z 541.368,A -85,B 0,C 180,E1 -7254.727,E2 -7254.727} C_VEL
LIN {X 0,Y 474.635,Z 541.362,A -85,B 0,C 180,E1 -7257.789,E2 -7257.789} C_VEL
LIN {X 0,Y 474.673,Z 541.483,A -85,B 0,C 180,E1 -7259.895,E2 -7259.895} C_VEL
LIN {X 0,Y 477.905,Z 556.154,A -85,B 0,C 180,E1 -7262.14,E2 -7262.14} C_VEL
LIN {X 0,Y 478.238,Z 559.846,A -85,B 0,C 180,E1 -7262.663,E2 -7262.663} C_VEL
LIN {X 0,Y 477.434,Z 578.742,A -85,B 0,C 180,E1 -7265.196,E2 -7265.196} C_VEL
LIN {X 0,Y 476.569,Z 602.958,A -85,B 0,C 180,E1 -7268.367,E2 -7268.367} C_VEL
LIN {X 0,Y 475.724,Z 628.904,A -85,B 0,C 180,E1 -7271.705,E2 -7271.705} C_VEL
LIN {X 0,Y 475.437,Z 640.699,A -85,B 0,C 180,E1 -7273.203,E2 -7273.203} C_VEL
LIN {X 0,Y 477.817,Z 664.314,A -85,B 0,C 180,E1 -7273.682,E2 -7273.682} C_VEL
LIN {X 0,Y 477.019,Z 752.271,A -85,B 0,C 180,E1 -7275.087,E2 -7275.087} C_VEL
LIN {X 0,Y 476.592,Z 771.4,A -85,B 0,C 180,E1 -7275.619,E2 -7275.619} C_VEL
LIN {X 0,Y 476.258,Z 784.673,A -85,B 0,C 180,E1 -7276.181,E2 -7276.181} C_VEL
LIN {X 0,Y 475.879,Z 796.57,A -85,B 0,C 180,E1 -7276.877,E2 -7276.877} C_VEL
LIN {X 0,Y 475.426,Z 807.602,A -85,B 0,C 180,E1 -7277.704,E2 -7277.704} C_VEL
LIN {X 0,Y 475.037,Z 818.154,A -85,B 0,C 180,E1 -7278.696,E2 -7278.696} C_VEL
LIN {X 0,Y 474.609,Z 827.311,A -85,B 0,C 180,E1 -7279.765,E2 -7279.765} C_VEL
LIN {X 0,Y 474.311,Z 836.213,A -85,B 0,C 180,E1 -7281.05,E2 -7281.05} C_VEL
LIN {X 0,Y 474.094,Z 843.333,A -85,B 0,C 180,E1 -7282.334,E2 -7282.334} C_VEL
LIN {X 0,Y 473.911,Z 849.551,A -85,B 0,C 180,E1 -7283.765,E2 -7283.765} C_VEL
LIN {X 0,Y 473.906,Z 853.413,A -85,B 0,C 180,E1 -7284.896,E2 -7284.896} C_VEL
LIN {X 0,Y 473.864,Z 855.744,A -85,B 0,C 180,E1 -7285.748,E2 -7285.748} C_VEL
LIN {X 0,Y 473.909,Z 857.644,A -85,B 0,C 180,E1 -7286.6,E2 -7286.6} C_VEL
LIN {X 0,Y 473.835,Z 859.076,A -85,B 0,C 180,E1 -7287.45,E2 -7287.45} C_VEL
LIN {X 0,Y 473.826,Z 860.086,A -85,B 0,C 180,E1 -7288.301,E2 -7288.301} C_VEL
LIN {X 0,Y 473.797,Z 860.702,A -85,B 0,C 180,E1 -7289.151,E2 -7289.151} C_VEL
LIN {X 0,Y 473.799,Z 860.923,A -85,B 0,C 180,E1 -7290.001,E2 -7290.001} C_VEL
LIN {X 0,Y 473.82,Z 860.083,A -85,B 0,C 180,E1 -7291.701,E2 -7291.701} C_VEL
LIN {X 0,Y 473.824,Z 859.072,A -85,B 0,C 180,E1 -7292.551,E2 -7292.551} C_VEL
LIN {X 0,Y 473.884,Z 857.639,A -85,B 0,C 180,E1 -7293.402,E2 -7293.402} C_VEL
LIN {X 0,Y 473.847,Z 854.652,A -85,B 0,C 180,E1 -7294.68,E2 -7294.68} C_VEL
LIN {X 0,Y 473.946,Z 850.598,A -85,B 0,C 180,E1 -7295.959,E2 -7295.959} C_VEL
LIN {X 0,Y 474.035,Z 844.333,A -85,B 0,C 180,E1 -7297.454,E2 -7297.454} C_VEL
LIN {X 0,Y 474.284,Z 837.497,A -85,B 0,C 180,E1 -7298.737,E2 -7298.737} C_VEL
LIN {X 0,Y 474.503,Z 830.506,A -85,B 0,C 180,E1 -7299.808,E2 -7299.808} C_VEL
LIN {X 0,Y 474.792,Z 822.052,A -85,B 0,C 180,E1 -7300.879,E2 -7300.879} C_VEL
LIN {X 0,Y 475.229,Z 811.561,A -85,B 0,C 180,E1 -7301.95,E2 -7301.95} C_VEL
LIN {X 0,Y 475.588,Z 801.145,A -85,B 0,C 180,E1 -7302.807,E2 -7302.807} C_VEL
LIN {X 0,Y 476.072,Z 789.637,A -85,B 0,C 180,E1 -7303.554,E2 -7303.554} C_VEL
LIN {X 0,Y 476.456,Z 777.631,A -85,B 0,C 180,E1 -7304.141,E2 -7304.141} C_VEL
LIN {X 0,Y 476.899,Z 763.358,A -85,B 0,C 180,E1 -7304.673,E2 -7304.673} C_VEL
LIN {X 0,Y 477.19,Z 750.434,A -85,B 0,C 180,E1 -7304.991,E2 -7304.991} C_VEL
LIN {X 0,Y 477.739,Z 663.699,A -85,B 0,C 180,E1 -7306.368,E2 -7306.368} C_VEL
LIN {X 0,Y 475.346,Z 643.8,A -85,B 0,C 180,E1 -7306.785,E2 -7306.785} C_VEL
LIN {X 0,Y 476.086,Z 619.409,A -85,B 0,C 180,E1 -7310.299,E2 -7310.299} C_VEL
LIN {X 0,Y 476.797,Z 599.362,A -85,B 0,C 180,E1 -7313.222,E2 -7313.222} C_VEL
LIN {X 0,Y 477.699,Z 577.718,A -85,B 0,C 180,E1 -7316.426,E2 -7316.426} C_VEL
LIN {X 0,Y 478.462,Z 560.619,A -85,B 0,C 180,E1 -7318.995,E2 -7318.995} C_VEL
LIN {X 0,Y 477.835,Z 555.614,A -85,B 0,C 180,E1 -7319.799,E2 -7319.799} C_VEL
LIN {X 0,Y 474.639,Z 541.364,A -85,B 0,C 180,E1 -7322.212,E2 -7322.212} C_VEL
LIN {X 0,Y 474.628,Z 541.365,A -85,B 0,C 180,E1 -7325.274,E2 -7325.274} C_VEL
LIN {X 0,Y 474.614,Z 541.363,A -85,B 0,C 180,E1 -7328.457,E2 -7328.457} C_VEL
LIN {X 0,Y 474.63,Z 541.366,A -85,B 0,C 180,E1 -7330.959,E2 -7330.959} C_VEL
LIN {X 0,Y 474.611,Z 541.356,A -85,B 0,C 180,E1 -7334.105,E2 -7334.105} C_VEL
LIN {X 0,Y 474.646,Z 541.362,A -85,B 0,C 180,E1 -7337.069,E2 -7337.069} C_VEL
LIN {X 0,Y 474.646,Z 541.357,A -85,B 0,C 180,E1 -7340.454,E2 -7340.454} C_VEL
LIN {X 0,Y 474.594,Z 541.362,A -85,B 0,C 180,E1 -7343.677,E2 -7343.677} C_VEL
LIN {X 0,Y 474.644,Z 541.359,A -85,B 0,C 180,E1 -7346.78,E2 -7346.78} C_VEL
LIN {X 0,Y 474.606,Z 541.361,A -85,B 0,C 180,E1 -7349.77,E2 -7349.77} C_VEL
LIN {X 0,Y 474.698,Z 541.351,A -85,B 0,C 180,E1 -7352.68,E2 -7352.68} C_VEL
LIN {X 0,Y 474.657,Z 541.353,A -85,B 0,C 180,E1 -7355.507,E2 -7355.507} C_VEL
LIN {X 0,Y 474.67,Z 541.359,A -85,B 0,C 180,E1 -7359.185,E2 -7359.185} C_VEL
LIN {X 0,Y 474.657,Z 541.348,A -85,B 0,C 180,E1 -7361.884,E2 -7361.884} C_VEL
LIN {X 0,Y 474.7,Z 541.348,A -85,B 0,C 180,E1 -7364.544,E2 -7364.544} C_VEL
LIN {X 0,Y 474.704,Z 541.345,A -85,B 0,C 180,E1 -7368.038,E2 -7368.038} C_VEL
LIN {X 0,Y 474.728,Z 541.347,A -85,B 0,C 180,E1 -7371.486,E2 -7371.486} C_VEL
LIN {X 0,Y 474.778,Z 541.342,A -85,B 0,C 180,E1 -7374.052,E2 -7374.052} C_VEL
LIN {X 0,Y 474.894,Z 541.32,A -85,B 0,C 180,E1 -7377.455,E2 -7377.455} C_VEL
LIN {X 0,Y 474.911,Z 541.328,A -85,B 0,C 180,E1 -7380,E2 -7380} C_VEL
LIN {X 0,Y 474.894,Z 541.324,A -85,B 0,C 180,E1 -7382.545,E2 -7382.545} C_VEL
LIN {X 0,Y 474.779,Z 541.339,A -85,B 0,C 180,E1 -7385.948,E2 -7385.948} C_VEL
LIN {X 0,Y 474.728,Z 541.347,A -85,B 0,C 180,E1 -7388.514,E2 -7388.514} C_VEL
LIN {X 0,Y 474.704,Z 541.345,A -85,B 0,C 180,E1 -7391.963,E2 -7391.963} C_VEL
LIN {X 0,Y 474.7,Z 541.352,A -85,B 0,C 180,E1 -7395.456,E2 -7395.456} C_VEL
LIN {X 0,Y 474.665,Z 541.346,A -85,B 0,C 180,E1 -7399.01,E2 -7399.01} C_VEL
LIN {X 0,Y 474.589,Z 541.367,A -85,B 0,C 180,E1 -7401.729,E2 -7401.729} C_VEL
LIN {X 0,Y 474.66,Z 541.351,A -85,B 0,C 180,E1 -7404.493,E2 -7404.493} C_VEL
LIN {X 0,Y 474.682,Z 541.352,A -85,B 0,C 180,E1 -7407.335,E2 -7407.335} C_VEL
LIN {X 0,Y 474.605,Z 541.362,A -85,B 0,C 180,E1 -7410.23,E2 -7410.23} C_VEL
LIN {X 0,Y 474.644,Z 541.358,A -85,B 0,C 180,E1 -7413.22,E2 -7413.22} C_VEL
LIN {X 0,Y 474.59,Z 541.37,A -85,B 0,C 180,E1 -7416.324,E2 -7416.324} C_VEL
LIN {X 0,Y 474.629,Z 541.36,A -85,B 0,C 180,E1 -7419.648,E2 -7419.648} C_VEL
LIN {X 0,Y 474.616,Z 541.358,A -85,B 0,C 180,E1 -7422.934,E2 -7422.934} C_VEL
LIN {X 0,Y 474.605,Z 541.366,A -85,B 0,C 180,E1 -7425.895,E2 -7425.895} C_VEL
LIN {X 0,Y 474.63,Z 541.361,A -85,B 0,C 180,E1 -7429.041,E2 -7429.041} C_VEL
LIN {X 0,Y 474.612,Z 541.36,A -85,B 0,C 180,E1 -7431.704,E2 -7431.704} C_VEL
LIN {X 0,Y 474.63,Z 541.365,A -85,B 0,C 180,E1 -7434.726,E2 -7434.726} C_VEL
LIN {X 0,Y 474.64,Z 541.362,A -85,B 0,C 180,E1 -7437.788,E2 -7437.788} C_VEL
LIN {X 0,Y 474.684,Z 541.358,A -85,B 0,C 180,E1 -7441.479,E2 -7441.479} C_VEL
LIN {X 0,Y 474.738,Z 541.572,A -85,B 0,C 180,E1 -7441.723,E2 -7441.723} C_VEL
LIN {X 0,Y 477.876,Z 556.129,A -85,B 0,C 180,E1 -7443.999,E2 -7443.999} C_VEL
LIN {X 0,Y 478.058,Z 561.313,A -85,B 0,C 180,E1 -7444.765,E2 -7444.765} C_VEL
LIN {X 0,Y 477.091,Z 584.542,A -85,B 0,C 180,E1 -7448.133,E2 -7448.133} C_VEL
LIN {X 0,Y 476.962,Z 586.803,A -85,B 0,C 180,E1 -7448.46,E2 -7448.46} C_VEL
LIN {X 0,Y 476.225,Z 590.676,A -85,B 0,C 180,E1 -7448.99,E2 -7448.99} C_VEL
LIN {X 0,Y 470.189,Z 603.903,A -85,B 0,C 180,E1 -7450.635,E2 -7450.635} C_VEL
LIN {X 0,Y 469.419,Z 607.842,A -85,B 0,C 180,E1 -7451.164,E2 -7451.164} C_VEL
LIN {X 0,Y 469.111,Z 621.77,A -85,B 0,C 180,E1 -7453.044,E2 -7453.044} C_VEL
LIN {X 0,Y 471.338,Z 636.523,A -85,B 0,C 180,E1 -7453.358,E2 -7453.358} C_VEL
LIN {X 0,Y 470.614,Z 732.13,A -85,B 0,C 180,E1 -7454.85,E2 -7454.85} C_VEL
LIN {X 0,Y 470.304,Z 745.398,A -85,B 0,C 180,E1 -7455.227,E2 -7455.227} C_VEL
LIN {X 0,Y 469.88,Z 757.879,A -85,B 0,C 180,E1 -7455.767,E2 -7455.767} C_VEL
LIN {X 0,Y 469.418,Z 769.948,A -85,B 0,C 180,E1 -7456.471,E2 -7456.471} C_VEL
LIN {X 0,Y 469.011,Z 781.373,A -85,B 0,C 180,E1 -7457.34,E2 -7457.34} C_VEL
LIN {X 0,Y 468.394,Z 792.655,A -85,B 0,C 180,E1 -7458.422,E2 -7458.422} C_VEL
LIN {X 0,Y 468.042,Z 800.893,A -85,B 0,C 180,E1 -7459.4,E2 -7459.4} C_VEL
LIN {X 0,Y 467.637,Z 808.499,A -85,B 0,C 180,E1 -7460.484,E2 -7460.484} C_VEL
LIN {X 0,Y 467.265,Z 815.923,A -85,B 0,C 180,E1 -7461.784,E2 -7461.784} C_VEL
LIN {X 0,Y 467.02,Z 822.844,A -85,B 0,C 180,E1 -7463.321,E2 -7463.321} C_VEL
LIN {X 0,Y 466.796,Z 827.936,A -85,B 0,C 180,E1 -7464.816,E2 -7464.816} C_VEL
LIN {X 0,Y 466.748,Z 830.214,A -85,B 0,C 180,E1 -7465.682,E2 -7465.682} C_VEL
LIN {X 0,Y 466.77,Z 832.07,A -85,B 0,C 180,E1 -7466.547,E2 -7466.547} C_VEL
LIN {X 0,Y 466.683,Z 833.495,A -85,B 0,C 180,E1 -7467.41,E2 -7467.41} C_VEL
LIN {X 0,Y 466.62,Z 835.109,A -85,B 0,C 180,E1 -7469.136,E2 -7469.136} C_VEL
LIN {X 0,Y 466.599,Z 835.346,A -85,B 0,C 180,E1 -7469.999,E2 -7469.999} C_VEL
LIN {X 0,Y 466.619,Z 835.159,A -85,B 0,C 180,E1 -7470.862,E2 -7470.862} C_VEL
LIN {X 0,Y 466.683,Z 833.613,A -85,B 0,C 180,E1 -7472.589,E2 -7472.589} C_VEL
LIN {X 0,Y 466.769,Z 832.252,A -85,B 0,C 180,E1 -7473.452,E2 -7473.452} C_VEL
LIN {X 0,Y 466.733,Z 829.394,A -85,B 0,C 180,E1 -7474.75,E2 -7474.75} C_VEL
LIN {X 0,Y 466.961,Z 825.502,A -85,B 0,C 180,E1 -7476.047,E2 -7476.047} C_VEL
LIN {X 0,Y 467.094,Z 820.469,A -85,B 0,C 180,E1 -7477.347,E2 -7477.347} C_VEL
LIN {X 0,Y 467.346,Z 814.123,A -85,B 0,C 180,E1 -7478.648,E2 -7478.648} C_VEL
LIN {X 0,Y 467.721,Z 806.227,A -85,B 0,C 180,E1 -7479.95,E2 -7479.95} C_VEL
LIN {X 0,Y 468.097,Z 798.159,A -85,B 0,C 180,E1 -7481.035,E2 -7481.035} C_VEL
LIN {X 0,Y 468.697,Z 788.267,A -85,B 0,C 180,E1 -7482.117,E2 -7482.117} C_VEL
LIN {X 0,Y 469.14,Z 777.028,A -85,B 0,C 180,E1 -7483.106,E2 -7483.106} C_VEL
LIN {X 0,Y 469.596,Z 766.299,A -85,B 0,C 180,E1 -7483.854,E2 -7483.854} C_VEL
LIN {X 0,Y 470.04,Z 754.145,A -85,B 0,C 180,E1 -7484.503,E2 -7484.503} C_VEL
LIN {X 0,Y 470.436,Z 740.75,A -85,B 0,C 180,E1 -7485.016,E2 -7485.016} C_VEL
LIN {X 0,Y 470.632,Z 728.634,A -85,B 0,C 180,E1 -7485.314,E2 -7485.314} C_VEL
LIN {X 0,Y 471.345,Z 638.007,A -85,B 0,C 180,E1 -7486.709,E2 -7486.709} C_VEL
LIN {X 0,Y 468.803,Z 622.457,A -85,B 0,C 180,E1 -7487.057,E2 -7487.057} C_VEL
LIN {X 0,Y 469.289,Z 603.738,A -85,B 0,C 180,E1 -7489.918,E2 -7489.918} C_VEL
LIN {X 0,Y 470.016,Z 584.014,A -85,B 0,C 180,E1 -7493.109,E2 -7493.109} C_VEL
LIN {X 0,Y 470.657,Z 567.307,A -85,B 0,C 180,E1 -7495.855,E2 -7495.855} C_VEL
LIN {X 0,Y 470.907,Z 558.456,A -85,B 0,C 180,E1 -7497.316,E2 -7497.316} C_VEL
LIN {X 0,Y 468.926,Z 548.146,A -85,B 0,C 180,E1 -7499.122,E2 -7499.122} C_VEL
LIN {X 0,Y 467.571,Z 542.245,A -85,B 0,C 180,E1 -7500.17,E2 -7500.17} C_VEL
LIN {X 0,Y 467.581,Z 542.243,A -85,B 0,C 180,E1 -7502.757,E2 -7502.757} C_VEL
LIN {X 0,Y 467.554,Z 542.241,A -85,B 0,C 180,E1 -7505.888,E2 -7505.888} C_VEL
LIN {X 0,Y 467.578,Z 542.239,A -85,B 0,C 180,E1 -7509.143,E2 -7509.143} C_VEL
LIN {X 0,Y 467.581,Z 542.237,A -85,B 0,C 180,E1 -7512.566,E2 -7512.566} C_VEL
LIN {X 0,Y 467.565,Z 542.239,A -85,B 0,C 180,E1 -7515.052,E2 -7515.052} C_VEL
LIN {X 0,Y 467.618,Z 542.24,A -85,B 0,C 180,E1 -7517.443,E2 -7517.443} C_VEL
LIN {X 0,Y 467.622,Z 542.236,A -85,B 0,C 180,E1 -7520.859,E2 -7520.859} C_VEL
LIN {X 0,Y 467.636,Z 542.287,A -85,B 0,C 180,E1 -7521.588,E2 -7521.588} C_VEL
LIN {X 0,Y 471.14,Z 553.216,A -85,B 0,C 180,E1 -7521.897,E2 -7521.897} C_VEL
LIN {X 0,Y 470.5,Z 622.415,A -85,B 0,C 180,E1 -7523.042,E2 -7523.042} C_VEL
LIN {X 0,Y 470.377,Z 635.386,A -85,B 0,C 180,E1 -7523.426,E2 -7523.426} C_VEL
LIN {X 0,Y 470.236,Z 648.086,A -85,B 0,C 180,E1 -7523.98,E2 -7523.98} C_VEL
LIN {X 0,Y 469.897,Z 660.403,A -85,B 0,C 180,E1 -7524.711,E2 -7524.711} C_VEL
LIN {X 0,Y 469.506,Z 671.937,A -85,B 0,C 180,E1 -7525.592,E2 -7525.592} C_VEL
LIN {X 0,Y 469.14,Z 682.134,A -85,B 0,C 180,E1 -7526.567,E2 -7526.567} C_VEL
LIN {X 0,Y 468.766,Z 690.833,A -85,B 0,C 180,E1 -7527.589,E2 -7527.589} C_VEL
LIN {X 0,Y 468.422,Z 699.134,A -85,B 0,C 180,E1 -7528.779,E2 -7528.779} C_VEL
LIN {X 0,Y 468.089,Z 706.357,A -85,B 0,C 180,E1 -7530.051,E2 -7530.051} C_VEL
LIN {X 0,Y 467.867,Z 711.941,A -85,B 0,C 180,E1 -7531.27,E2 -7531.27} C_VEL
LIN {X 0,Y 467.676,Z 717.463,A -85,B 0,C 180,E1 -7532.82,E2 -7532.82} C_VEL
LIN {X 0,Y 467.48,Z 721.541,A -85,B 0,C 180,E1 -7534.422,E2 -7534.422} C_VEL
LIN {X 0,Y 467.387,Z 724.182,A -85,B 0,C 180,E1 -7536.046,E2 -7536.046} C_VEL
LIN {X 0,Y 467.346,Z 725.012,A -85,B 0,C 180,E1 -7536.984,E2 -7536.984} C_VEL
LIN {X 0,Y 467.347,Z 725.408,A -85,B 0,C 180,E1 -7537.917,E2 -7537.917} C_VEL
LIN {X 0,Y 467.378,Z 725.322,A -85,B 0,C 180,E1 -7538.845,E2 -7538.845} C_VEL
LIN {X 0,Y 467.407,Z 724.764,A -85,B 0,C 180,E1 -7539.767,E2 -7539.767} C_VEL
LIN {X 0,Y 467.524,Z 722.902,A -85,B 0,C 180,E1 -7541.265,E2 -7541.265} C_VEL
LIN {X 0,Y 467.765,Z 719.215,A -85,B 0,C 180,E1 -7542.963,E2 -7542.963} C_VEL
LIN {X 0,Y 467.975,Z 714.997,A -85,B 0,C 180,E1 -7544.316,E2 -7544.316} C_VEL
LIN {X 0,Y 468.221,Z 709.55,A -85,B 0,C 180,E1 -7545.661,E2 -7545.661} C_VEL
LIN {X 0,Y 468.635,Z 702.069,A -85,B 0,C 180,E1 -7547.1,E2 -7547.1} C_VEL
LIN {X 0,Y 468.99,Z 693.999,A -85,B 0,C 180,E1 -7548.328,E2 -7548.328} C_VEL
LIN {X 0,Y 469.421,Z 684.112,A -85,B 0,C 180,E1 -7549.541,E2 -7549.541} C_VEL
LIN {X 0,Y 469.834,Z 673.994,A -85,B 0,C 180,E1 -7550.529,E2 -7550.529} C_VEL
LIN {X 0,Y 470.19,Z 662.809,A -85,B 0,C 180,E1 -7551.404,E2 -7551.404} C_VEL
LIN {X 0,Y 470.545,Z 651.158,A -85,B 0,C 180,E1 -7552.113,E2 -7552.113} C_VEL
LIN {X 0,Y 470.702,Z 639.264,A -85,B 0,C 180,E1 -7552.655,E2 -7552.655} C_VEL
LIN {X 0,Y 470.737,Z 626.497,A -85,B 0,C 180,E1 -7553.059,E2 -7553.059} C_VEL
LIN {X 0,Y 470.875,Z 600.827,A -85,B 0,C 180,E1 -7553.519,E2 -7553.519} C_VEL
LIN {X 0,Y 471.395,Z 552.568,A -85,B 0,C 180,E1 -7554.331,E2 -7554.331} C_VEL
LIN {X 0,Y 467.727,Z 542.236,A -85,B 0,C 180,E1 -7554.665,E2 -7554.665} C_VEL
LIN {X 0,Y 467.857,Z 542.206,A -85,B 0,C 180,E1 -7557.417,E2 -7557.417} C_VEL
LIN {X 0,Y 467.871,Z 542.206,A -85,B 0,C 180,E1 -7560,E2 -7560} C_VEL
LIN {X 0,Y 467.851,Z 542.212,A -85,B 0,C 180,E1 -7562.583,E2 -7562.583} C_VEL
LIN {X 0,Y 467.743,Z 542.218,A -85,B 0,C 180,E1 -7566.037,E2 -7566.037} C_VEL
LIN {X 0,Y 467.672,Z 542.232,A -85,B 0,C 180,E1 -7568.643,E2 -7568.643} C_VEL
LIN {X 0,Y 467.672,Z 542.228,A -85,B 0,C 180,E1 -7572.145,E2 -7572.145} C_VEL
LIN {X 0,Y 467.638,Z 542.227,A -85,B 0,C 180,E1 -7575.886,E2 -7575.886} C_VEL
LIN {X 0,Y 467.613,Z 542.235,A -85,B 0,C 180,E1 -7579.308,E2 -7579.308} C_VEL
LIN {X 0,Y 467.525,Z 542.245,A -85,B 0,C 180,E1 -7582.074,E2 -7582.074} C_VEL
LIN {X 0,Y 467.594,Z 542.242,A -85,B 0,C 180,E1 -7584.888,E2 -7584.888} C_VEL
LIN {X 0,Y 467.619,Z 542.232,A -85,B 0,C 180,E1 -7587.769,E2 -7587.769} C_VEL
LIN {X 0,Y 467.564,Z 542.245,A -85,B 0,C 180,E1 -7591.047,E2 -7591.047} C_VEL
LIN {X 0,Y 467.582,Z 542.239,A -85,B 0,C 180,E1 -7594.244,E2 -7594.244} C_VEL
LIN {X 0,Y 467.545,Z 542.243,A -85,B 0,C 180,E1 -7597.188,E2 -7597.188} C_VEL
LIN {X 0,Y 467.591,Z 542.238,A -85,B 0,C 180,E1 -7600.263,E2 -7600.263} C_VEL
LIN {X 0,Y 467.612,Z 542.239,A -85,B 0,C 180,E1 -7602.572,E2 -7602.572} C_VEL
LIN {X 0,Y 467.569,Z 542.242,A -85,B 0,C 180,E1 -7606.177,E2 -7606.177} C_VEL
LIN {X 0,Y 467.584,Z 542.243,A -85,B 0,C 180,E1 -7608.723,E2 -7608.723} C_VEL
LIN {X 0,Y 467.574,Z 542.242,A -85,B 0,C 180,E1 -7611.408,E2 -7611.408} C_VEL
LIN {X 0,Y 467.56,Z 542.246,A -85,B 0,C 180,E1 -7614.261,E2 -7614.261} C_VEL
LIN {X 0,Y 467.579,Z 542.244,A -85,B 0,C 180,E1 -7617.322,E2 -7617.322} C_VEL
LIN {X 0,Y 467.599,Z 542.369,A -85,B 0,C 180,E1 -7619.613,E2 -7619.613} C_VEL
LIN {X 0,Y 470.694,Z 555.971,A -85,B 0,C 180,E1 -7621.756,E2 -7621.756} C_VEL
LIN {X 0,Y 471.361,Z 560.783,A -85,B 0,C 180,E1 -7622.471,E2 -7622.471} C_VEL
LIN {X 0,Y 470.509,Z 579.614,A -85,B 0,C 180,E1 -7625.042,E2 -7625.042} C_VEL
LIN {X 0,Y 469.54,Z 604.456,A -85,B 0,C 180,E1 -7628.363,E2 -7628.363} C_VEL
LIN {X 0,Y 468.642,Z 631.3,A -85,B 0,C 180,E1 -7631.871,E2 -7631.871} C_VEL
LIN {X 0,Y 468.415,Z 639.85,A -85,B 0,C 180,E1 -7632.947,E2 -7632.947} C_VEL
LIN {X 0,Y 470.963,Z 665.214,A -85,B 0,C 180,E1 -7633.469,E2 -7633.469} C_VEL
LIN {X 0,Y 470.118,Z 751.965,A -85,B 0,C 180,E1 -7634.891,E2 -7634.891} C_VEL
LIN {X 0,Y 469.782,Z 768.994,A -85,B 0,C 180,E1 -7635.323,E2 -7635.323} C_VEL
LIN {X 0,Y 469.441,Z 781.159,A -85,B 0,C 180,E1 -7635.81,E2 -7635.81} C_VEL
LIN {X 0,Y 469.056,Z 793.068,A -85,B 0,C 180,E1 -7636.462,E2 -7636.462} C_VEL
LIN {X 0,Y 468.605,Z 804.017,A -85,B 0,C 180,E1 -7637.234,E2 -7637.234} C_VEL
LIN {X 0,Y 468.147,Z 814.791,A -85,B 0,C 180,E1 -7638.198,E2 -7638.198} C_VEL
LIN {X 0,Y 467.749,Z 823.675,A -85,B 0,C 180,E1 -7639.176,E2 -7639.176} C_VEL
LIN {X 0,Y 467.436,Z 831.824,A -85,B 0,C 180,E1 -7640.263,E2 -7640.263} C_VEL
LIN {X 0,Y 467.154,Z 839.794,A -85,B 0,C 180,E1 -7641.566,E2 -7641.566} C_VEL
LIN {X 0,Y 466.953,Z 845.167,A -85,B 0,C 180,E1 -7642.651,E2 -7642.651} C_VEL
LIN {X 0,Y 466.842,Z 850.413,A -85,B 0,C 180,E1 -7643.952,E2 -7643.952} C_VEL
LIN {X 0,Y 466.776,Z 854.466,A -85,B 0,C 180,E1 -7645.251,E2 -7645.251} C_VEL
LIN {X 0,Y 466.816,Z 857.452,A -85,B 0,C 180,E1 -7646.548,E2 -7646.548} C_VEL
LIN {X 0,Y 466.752,Z 858.884,A -85,B 0,C 180,E1 -7647.412,E2 -7647.412} C_VEL
LIN {X 0,Y 466.721,Z 860.51,A -85,B 0,C 180,E1 -7649.138,E2 -7649.138} C_VEL
LIN {X 0,Y 466.72,Z 860.731,A -85,B 0,C 180,E1 -7650.001,E2 -7650.001} C_VEL
LIN {X 0,Y 466.722,Z 859.891,A -85,B 0,C 180,E1 -7651.726,E2 -7651.726} C_VEL
LIN {X 0,Y 466.74,Z 858.88,A -85,B 0,C 180,E1 -7652.59,E2 -7652.59} C_VEL
LIN {X 0,Y 466.793,Z 857.447,A -85,B 0,C 180,E1 -7653.453,E2 -7653.453} C_VEL
LIN {X 0,Y 466.769,Z 854.461,A -85,B 0,C 180,E1 -7654.751,E2 -7654.751} C_VEL
LIN {X 0,Y 466.849,Z 850.408,A -85,B 0,C 180,E1 -7656.05,E2 -7656.05} C_VEL
LIN {X 0,Y 466.981,Z 844.145,A -85,B 0,C 180,E1 -7657.568,E2 -7657.568} C_VEL
LIN {X 0,Y 467.22,Z 837.312,A -85,B 0,C 180,E1 -7658.87,E2 -7658.87} C_VEL
LIN {X 0,Y 467.453,Z 830.323,A -85,B 0,C 180,E1 -7659.957,E2 -7659.957} C_VEL
LIN {X 0,Y 467.8,Z 821.873,A -85,B 0,C 180,E1 -7661.044,E2 -7661.044} C_VEL
LIN {X 0,Y 468.269,Z 811.388,A -85,B 0,C 180,E1 -7662.13,E2 -7662.13} C_VEL
LIN {X 0,Y 468.66,Z 800.978,A -85,B 0,C 180,E1 -7663,E2 -7663} C_VEL
LIN {X 0,Y 469.136,Z 789.479,A -85,B 0,C 180,E1 -7663.758,E2 -7663.758} C_VEL
LIN {X 0,Y 469.563,Z 777.49,A -85,B 0,C 180,E1 -7664.353,E2 -7664.353} C_VEL
LIN {X 0,Y 469.849,Z 765.35,A -85,B 0,C 180,E1 -7664.787,E2 -7664.787} C_VEL
LIN {X 0,Y 470.211,Z 751.734,A -85,B 0,C 180,E1 -7665.163,E2 -7665.163} C_VEL
LIN {X 0,Y 470.996,Z 665.224,A -85,B 0,C 180,E1 -7666.562,E2 -7666.562} C_VEL
LIN {X 0,Y 468.303,Z 642.917,A -85,B 0,C 180,E1 -7667.045,E2 -7667.045} C_VEL
LIN {X 0,Y 469.056,Z 620.095,A -85,B 0,C 180,E1 -7670.388,E2 -7670.388} C_VEL
LIN {X 0,Y 469.837,Z 600.076,A -85,B 0,C 180,E1 -7673.353,E2 -7673.353} C_VEL
LIN {X 0,Y 470.775,Z 578.405,A -85,B 0,C 180,E1 -7676.607,E2 -7676.607} C_VEL
LIN {X 0,Y 471.565,Z 561.344,A -85,B 0,C 180,E1 -7679.216,E2 -7679.216} C_VEL
LIN {X 0,Y 470.323,Z 554.373,A -85,B 0,C 180,E1 -7680.377,E2 -7680.377} C_VEL
LIN {X 0,Y 467.596,Z 542.242,A -85,B 0,C 180,E1 -7682.502,E2 -7682.502} C_VEL
LIN {X 0,Y 467.563,Z 542.242,A -85,B 0,C 180,E1 -7685.739,E2 -7685.739} C_VEL
LIN {X 0,Y 467.585,Z 542.244,A -85,B 0,C 180,E1 -7689.145,E2 -7689.145} C_VEL
LIN {X 0,Y 467.588,Z 542.239,A -85,B 0,C 180,E1 -7692.567,E2 -7692.567} C_VEL
LIN {X 0,Y 467.572,Z 542.241,A -85,B 0,C 180,E1 -7695.053,E2 -7695.053} C_VEL
LIN {X 0,Y 467.59,Z 542.235,A -85,B 0,C 180,E1 -7697.44,E2 -7697.44} C_VEL
LIN {X 0,Y 467.584,Z 542.24,A -85,B 0,C 180,E1 -7700.855,E2 -7700.855} C_VEL
LIN {X 0,Y 467.564,Z 542.235,A -85,B 0,C 180,E1 -7704.26,E2 -7704.26} C_VEL
LIN {X 0,Y 467.583,Z 542.24,A -85,B 0,C 180,E1 -7707.321,E2 -7707.321} C_VEL
LIN {X 0,Y 467.57,Z 542.236,A -85,B 0,C 180,E1 -7710.667,E2 -7710.667} C_VEL
LIN {X 0,Y 467.617,Z 542.239,A -85,B 0,C 180,E1 -7713.2,E2 -7713.2} C_VEL
LIN {X 0,Y 467.593,Z 542.23,A -85,B 0,C 180,E1 -7716.468,E2 -7716.468} C_VEL
LIN {X 0,Y 467.622,Z 542.232,A -85,B 0,C 180,E1 -7719.777,E2 -7719.777} C_VEL
LIN {X 0,Y 467.609,Z 542.223,A -85,B 0,C 180,E1 -7722.507,E2 -7722.507} C_VEL
LIN {X 0,Y 467.609,Z 542.236,A -85,B 0,C 180,E1 -7725.197,E2 -7725.197} C_VEL
LIN {X 0,Y 467.655,Z 542.225,A -85,B 0,C 180,E1 -7727.855,E2 -7727.855} C_VEL
LIN {X 0,Y 467.682,Z 542.222,A -85,B 0,C 180,E1 -7731.357,E2 -7731.357} C_VEL
LIN {X 0,Y 467.743,Z 542.219,A -85,B 0,C 180,E1 -7733.963,E2 -7733.963} C_VEL
LIN {X 0,Y 467.859,Z 542.196,A -85,B 0,C 180,E1 -7737.417,E2 -7737.417} C_VEL
LIN {X 0,Y 467.881,Z 542.203,A -85,B 0,C 180,E1 -7740,E2 -7740} C_VEL
LIN {X 0,Y 467.859,Z 542.2,A -85,B 0,C 180,E1 -7742.583,E2 -7742.583} C_VEL
LIN {X 0,Y 467.743,Z 542.216,A -85,B 0,C 180,E1 -7746.037,E2 -7746.037} C_VEL
LIN {X 0,Y 467.682,Z 542.224,A -85,B 0,C 180,E1 -7748.643,E2 -7748.643} C_VEL
LIN {X 0,Y 467.655,Z 542.221,A -85,B 0,C 180,E1 -7752.146,E2 -7752.146} C_VEL
LIN {X 0,Y 467.639,Z 542.235,A -85,B 0,C 180,E1 -7755.695,E2 -7755.695} C_VEL
LIN {X 0,Y 467.617,Z 542.224,A -85,B 0,C 180,E1 -7758.765,E2 -7758.765} C_VEL
LIN {X 0,Y 467.581,Z 542.236,A -85,B 0,C 180,E1 -7761.268,E2 -7761.268} C_VEL
LIN {X 0,Y 467.574,Z 542.241,A -85,B 0,C 180,E1 -7763.943,E2 -7763.943} C_VEL
LIN {X 0,Y 467.617,Z 542.232,A -85,B 0,C 180,E1 -7766.8,E2 -7766.8} C_VEL
LIN {X 0,Y 467.554,Z 542.244,A -85,B 0,C 180,E1 -7769.738,E2 -7769.738} C_VEL
LIN {X 0,Y 467.584,Z 542.239,A -85,B 0,C 180,E1 -7772.758,E2 -7772.758} C_VEL
LIN {X 0,Y 467.554,Z 542.241,A -85,B 0,C 180,E1 -7775.89,E2 -7775.89} C_VEL
LIN {X 0,Y 467.584,Z 542.236,A -85,B 0,C 180,E1 -7779.145,E2 -7779.145} C_VEL
LIN {X 0,Y 467.588,Z 542.237,A -85,B 0,C 180,E1 -7782.567,E2 -7782.567} C_VEL
LIN {X 0,Y 467.567,Z 542.239,A -85,B 0,C 180,E1 -7785.053,E2 -7785.053} C_VEL
LIN {X 0,Y 467.578,Z 542.24,A -85,B 0,C 180,E1 -7788.597,E2 -7788.597} C_VEL
LIN {X 0,Y 467.564,Z 542.237,A -85,B 0,C 180,E1 -7791.409,E2 -7791.409} C_VEL
LIN {X 0,Y 467.564,Z 542.246,A -85,B 0,C 180,E1 -7794.261,E2 -7794.261} C_VEL
LIN {X 0,Y 467.585,Z 542.24,A -85,B 0,C 180,E1 -7797.321,E2 -7797.321} C_VEL
LIN {X 0,Y 467.574,Z 542.248,A -85,B 0,C 180,E1 -7800.667,E2 -7800.667} C_VEL
LIN {X 0,Y 467.637,Z 542.264,A -85,B 0,C 180,E1 -7801.438,E2 -7801.438} C_VEL
LIN {X 0,Y 471.101,Z 558.335,A -85,B 0,C 180,E1 -7803.982,E2 -7803.982} C_VEL
LIN {X 0,Y 471.12,Z 564.161,A -85,B 0,C 180,E1 -7804.839,E2 -7804.839} C_VEL
LIN {X 0,Y 470.15,Z 586.119,A -85,B 0,C 180,E1 -7808.055,E2 -7808.055} C_VEL
LIN {X 0,Y 469.419,Z 607.842,A -85,B 0,C 180,E1 -7811.164,E2 -7811.164} C_VEL
LIN {X 0,Y 468.635,Z 611.066,A -85,B 0,C 180,E1 -7811.562,E2 -7811.562} C_VEL
LIN {X 0,Y 466.86,Z 614.279,A -85,B 0,C 180,E1 -7811.923,E2 -7811.923} C_VEL
LIN {X 0,Y 462.484,Z 621.175,A -85,B 0,C 180,E1 -7812.703,E2 -7812.703} C_VEL
LIN {X 0,Y 462.366,Z 622.872,A -85,B 0,C 180,E1 -7812.805,E2 -7812.805} C_VEL
LIN {X 0,Y 464.547,Z 637.599,A -85,B 0,C 180,E1 -7813.123,E2 -7813.123} C_VEL
LIN {X 0,Y 463.768,Z 732.238,A -85,B 0,C 180,E1 -7814.621,E2 -7814.621} C_VEL
LIN {X 0,Y 463.464,Z 745.548,A -85,B 0,C 180,E1 -7815.004,E2 -7815.004} C_VEL
LIN {X 0,Y 463.017,Z 758.044,A -85,B 0,C 180,E1 -7815.552,E2 -7815.552} C_VEL
LIN {X 0,Y 462.527,Z 770.122,A -85,B 0,C 180,E1 -7816.266,E2 -7816.266} C_VEL
LIN {X 0,Y 462.089,Z 781.56,A -85,B 0,C 180,E1 -7817.148,E2 -7817.148} C_VEL
LIN {X 0,Y 461.459,Z 792.84,A -85,B 0,C 180,E1 -7818.246,E2 -7818.246} C_VEL
LIN {X 0,Y 461.063,Z 801.081,A -85,B 0,C 180,E1 -7819.238,E2 -7819.238} C_VEL
LIN {X 0,Y 460.638,Z 808.688,A -85,B 0,C 180,E1 -7820.338,E2 -7820.338} C_VEL
LIN {X 0,Y 460.236,Z 816.114,A -85,B 0,C 180,E1 -7821.658,E2 -7821.658} C_VEL
LIN {X 0,Y 459.943,Z 822.08,A -85,B 0,C 180,E1 -7822.978,E2 -7822.978} C_VEL
LIN {X 0,Y 459.871,Z 826.795,A -85,B 0,C 180,E1 -7824.298,E2 -7824.298} C_VEL
LIN {X 0,Y 459.654,Z 830.407,A -85,B 0,C 180,E1 -7825.615,E2 -7825.615} C_VEL
LIN {X 0,Y 459.683,Z 832.264,A -85,B 0,C 180,E1 -7826.493,E2 -7826.493} C_VEL
LIN {X 0,Y 459.607,Z 833.688,A -85,B 0,C 180,E1 -7827.37,E2 -7827.37} C_VEL
LIN {X 0,Y 459.523,Z 835.302,A -85,B 0,C 180,E1 -7829.123,E2 -7829.123} C_VEL
LIN {X 0,Y 459.53,Z 835.539,A -85,B 0,C 180,E1 -7829.999,E2 -7829.999} C_VEL
LIN {X 0,Y 459.523,Z 835.351,A -85,B 0,C 180,E1 -7830.876,E2 -7830.876} C_VEL
LIN {X 0,Y 459.607,Z 833.804,A -85,B 0,C 180,E1 -7832.629,E2 -7832.629} C_VEL
LIN {X 0,Y 459.683,Z 832.443,A -85,B 0,C 180,E1 -7833.505,E2 -7833.505} C_VEL
LIN {X 0,Y 459.661,Z 829.584,A -85,B 0,C 180,E1 -7834.823,E2 -7834.823} C_VEL
LIN {X 0,Y 459.888,Z 825.69,A -85,B 0,C 180,E1 -7836.14,E2 -7836.14} C_VEL
LIN {X 0,Y 460.039,Z 820.656,A -85,B 0,C 180,E1 -7837.46,E2 -7837.46} C_VEL
LIN {X 0,Y 460.331,Z 814.307,A -85,B 0,C 180,E1 -7838.781,E2 -7838.781} C_VEL
LIN {X 0,Y 460.71,Z 806.409,A -85,B 0,C 180,E1 -7840.103,E2 -7840.103} C_VEL
LIN {X 0,Y 461.136,Z 798.338,A -85,B 0,C 180,E1 -7841.204,E2 -7841.204} C_VEL
LIN {X 0,Y 461.759,Z 788.44,A -85,B 0,C 180,E1 -7842.302,E2 -7842.302} C_VEL
LIN {X 0,Y 462.243,Z 776.918,A -85,B 0,C 180,E1 -7843.327,E2 -7843.327} C_VEL
LIN {X 0,Y 462.708,Z 766.456,A -85,B 0,C 180,E1 -7844.064,E2 -7844.064} C_VEL
LIN {X 0,Y 463.185,Z 754.284,A -85,B 0,C 180,E1 -7844.722,E2 -7844.722} C_VEL
LIN {X 0,Y 463.603,Z 740.861,A -85,B 0,C 180,E1 -7845.243,E2 -7845.243} C_VEL
LIN {X 0,Y 463.8,Z 728.663,A -85,B 0,C 180,E1 -7845.545,E2 -7845.545} C_VEL
LIN {X 0,Y 464.559,Z 638.512,A -85,B 0,C 180,E1 -7846.953,E2 -7846.953} C_VEL
LIN {X 0,Y 461.857,Z 622.584,A -85,B 0,C 180,E1 -7847.318,E2 -7847.318} C_VEL
LIN {X 0,Y 462.313,Z 606.609,A -85,B 0,C 180,E1 -7849.769,E2 -7849.769} C_VEL
LIN {X 0,Y 462.972,Z 588.049,A -85,B 0,C 180,E1 -7852.773,E2 -7852.773} C_VEL
LIN {X 0,Y 463.768,Z 569.615,A -85,B 0,C 180,E1 -7855.827,E2 -7855.827} C_VEL
LIN {X 0,Y 463.982,Z 559.498,A -85,B 0,C 180,E1 -7857.514,E2 -7857.514} C_VEL
LIN {X 0,Y 461.405,Z 546.903,A -85,B 0,C 180,E1 -7859.748,E2 -7859.748} C_VEL
LIN {X 0,Y 460.533,Z 543.122,A -85,B 0,C 180,E1 -7860.427,E2 -7860.427} C_VEL
LIN {X 0,Y 460.527,Z 543.119,A -85,B 0,C 180,E1 -7863.324,E2 -7863.324} C_VEL
LIN {X 0,Y 460.476,Z 543.123,A -85,B 0,C 180,E1 -7866.528,E2 -7866.528} C_VEL
LIN {X 0,Y 460.554,Z 543.114,A -85,B 0,C 180,E1 -7869.858,E2 -7869.858} C_VEL
LIN {X 0,Y 460.512,Z 543.117,A -85,B 0,C 180,E1 -7872.9,E2 -7872.9} C_VEL
LIN {X 0,Y 460.518,Z 543.12,A -85,B 0,C 180,E1 -7875.828,E2 -7875.828} C_VEL
LIN {X 0,Y 460.537,Z 543.119,A -85,B 0,C 180,E1 -7878.989,E2 -7878.989} C_VEL
LIN {X 0,Y 460.565,Z 543.119,A -85,B 0,C 180,E1 -7881.328,E2 -7881.328} C_VEL
LIN {X 0,Y 464.175,Z 553.816,A -85,B 0,C 180,E1 -7881.665,E2 -7881.665} C_VEL
LIN {X 0,Y 463.629,Z 623.028,A -85,B 0,C 180,E1 -7882.835,E2 -7882.835} C_VEL
LIN {X 0,Y 463.519,Z 635.566,A -85,B 0,C 180,E1 -7883.206,E2 -7883.206} C_VEL
LIN {X 0,Y 463.396,Z 647.807,A -85,B 0,C 180,E1 -7883.737,E2 -7883.737} C_VEL
LIN {X 0,Y 463.082,Z 659.011,A -85,B 0,C 180,E1 -7884.38,E2 -7884.38} C_VEL
LIN {X 0,Y 462.721,Z 670.193,A -85,B 0,C 180,E1 -7885.204,E2 -7885.204} C_VEL
LIN {X 0,Y 462.281,Z 680.995,A -85,B 0,C 180,E1 -7886.204,E2 -7886.204} C_VEL
LIN {X 0,Y 461.872,Z 690.615,A -85,B 0,C 180,E1 -7887.304,E2 -7887.304} C_VEL
LIN {X 0,Y 461.529,Z 699.127,A -85,B 0,C 180,E1 -7888.509,E2 -7888.509} C_VEL
LIN {X 0,Y 461.152,Z 706.565,A -85,B 0,C 180,E1 -7889.806,E2 -7889.806} C_VEL
LIN {X 0,Y 460.85,Z 713.339,A -85,B 0,C 180,E1 -7891.29,E2 -7891.29} C_VEL
LIN {X 0,Y 460.661,Z 718.449,A -85,B 0,C 180,E1 -7892.762,E2 -7892.762} C_VEL
LIN {X 0,Y 460.506,Z 722.16,A -85,B 0,C 180,E1 -7894.211,E2 -7894.211} C_VEL
LIN {X 0,Y 460.387,Z 724.693,A -85,B 0,C 180,E1 -7895.659,E2 -7895.659} C_VEL
LIN {X 0,Y 460.354,Z 725.768,A -85,B 0,C 180,E1 -7896.613,E2 -7896.613} C_VEL
LIN {X 0,Y 460.325,Z 726.32,A -85,B 0,C 180,E1 -7897.562,E2 -7897.562} C_VEL
LIN {X 0,Y 460.358,Z 726.409,A -85,B 0,C 180,E1 -7898.626,E2 -7898.626} C_VEL
LIN {X 0,Y 460.372,Z 726.081,A -85,B 0,C 180,E1 -7899.444,E2 -7899.444} C_VEL
LIN {X 0,Y 460.509,Z 724.254,A -85,B 0,C 180,E1 -7901.116,E2 -7901.116} C_VEL
LIN {X 0,Y 460.716,Z 721.152,A -85,B 0,C 180,E1 -7902.695,E2 -7902.695} C_VEL
LIN {X 0,Y 460.921,Z 717.247,A -85,B 0,C 180,E1 -7904.07,E2 -7904.07} C_VEL
LIN {X 0,Y 461.24,Z 711.12,A -85,B 0,C 180,E1 -7905.664,E2 -7905.664} C_VEL
LIN {X 0,Y 461.617,Z 704.511,A -85,B 0,C 180,E1 -7906.996,E2 -7906.996} C_VEL
LIN {X 0,Y 461.986,Z 697.448,A -85,B 0,C 180,E1 -7908.149,E2 -7908.149} C_VEL
LIN {X 0,Y 462.402,Z 689.08,A -85,B 0,C 180,E1 -7909.27,E2 -7909.27} C_VEL
LIN {X 0,Y 462.818,Z 678.731,A -85,B 0,C 180,E1 -7910.384,E2 -7910.384} C_VEL
LIN {X 0,Y 463.257,Z 668.428,A -85,B 0,C 180,E1 -7911.274,E2 -7911.274} C_VEL
LIN {X 0,Y 463.615,Z 657.157,A -85,B 0,C 180,E1 -7912.049,E2 -7912.049} C_VEL
LIN {X 0,Y 463.83,Z 644.398,A -85,B 0,C 180,E1 -7912.709,E2 -7912.709} C_VEL
LIN {X 0,Y 463.919,Z 631.803,A -85,B 0,C 180,E1 -7913.176,E2 -7913.176} C_VEL
LIN {X 0,Y 463.977,Z 618.542,A -85,B 0,C 180,E1 -7913.477,E2 -7913.477} C_VEL
LIN {X 0,Y 464.545,Z 553.794,A -85,B 0,C 180,E1 -7914.591,E2 -7914.591} C_VEL
LIN {X 0,Y 460.656,Z 543.107,A -85,B 0,C 180,E1 -7914.967,E2 -7914.967} C_VEL
LIN {X 0,Y 460.823,Z 543.083,A -85,B 0,C 180,E1 -7917.378,E2 -7917.378} C_VEL
LIN {X 0,Y 460.842,Z 543.081,A -85,B 0,C 180,E1 -7920,E2 -7920} C_VEL
LIN {X 0,Y 460.816,Z 543.089,A -85,B 0,C 180,E1 -7922.622,E2 -7922.622} C_VEL
LIN {X 0,Y 460.708,Z 543.095,A -85,B 0,C 180,E1 -7926.13,E2 -7926.13} C_VEL
LIN {X 0,Y 460.619,Z 543.112,A -85,B 0,C 180,E1 -7928.776,E2 -7928.776} C_VEL
LIN {X 0,Y 460.623,Z 543.108,A -85,B 0,C 180,E1 -7932.457,E2 -7932.457} C_VEL
LIN {X 0,Y 460.589,Z 543.105,A -85,B 0,C 180,E1 -7935.998,E2 -7935.998} C_VEL
LIN {X 0,Y 460.561,Z 543.118,A -85,B 0,C 180,E1 -7938.903,E2 -7938.903} C_VEL
LIN {X 0,Y 460.505,Z 543.12,A -85,B 0,C 180,E1 -7941.486,E2 -7941.486} C_VEL
LIN {X 0,Y 460.533,Z 543.118,A -85,B 0,C 180,E1 -7944.333,E2 -7944.333} C_VEL
LIN {X 0,Y 460.575,Z 543.112,A -85,B 0,C 180,E1 -7947.244,E2 -7947.244} C_VEL
LIN {X 0,Y 460.518,Z 543.119,A -85,B 0,C 180,E1 -7950.24,E2 -7950.24} C_VEL
LIN {X 0,Y 460.521,Z 543.119,A -85,B 0,C 180,E1 -7953.326,E2 -7953.326} C_VEL
LIN {X 0,Y 460.472,Z 543.128,A -85,B 0,C 180,E1 -7956.53,E2 -7956.53} C_VEL
LIN {X 0,Y 460.572,Z 543.111,A -85,B 0,C 180,E1 -7959.858,E2 -7959.858} C_VEL
LIN {X 0,Y 460.536,Z 543.12,A -85,B 0,C 180,E1 -7962.905,E2 -7962.905} C_VEL
LIN {X 0,Y 460.518,Z 543.12,A -85,B 0,C 180,E1 -7965.83,E2 -7965.83} C_VEL
LIN {X 0,Y 460.538,Z 543.12,A -85,B 0,C 180,E1 -7968.991,E2 -7968.991} C_VEL
LIN {X 0,Y 460.543,Z 543.12,A -85,B 0,C 180,E1 -7971.27,E2 -7971.27} C_VEL
LIN {X 0,Y 460.511,Z 543.127,A -85,B 0,C 180,E1 -7974.556,E2 -7974.556} C_VEL
LIN {X 0,Y 460.529,Z 543.12,A -85,B 0,C 180,E1 -7977.717,E2 -7977.717} C_VEL
LIN {X 0,Y 460.567,Z 543.233,A -85,B 0,C 180,E1 -7979.322,E2 -7979.322} C_VEL
LIN {X 0,Y 463.69,Z 556.895,A -85,B 0,C 180,E1 -7981.533,E2 -7981.533} C_VEL
LIN {X 0,Y 464.504,Z 561.767,A -85,B 0,C 180,E1 -7982.275,E2 -7982.275} C_VEL
LIN {X 0,Y 463.505,Z 581.812,A -85,B 0,C 180,E1 -7985.071,E2 -7985.071} C_VEL
LIN {X 0,Y 462.479,Z 606.512,A -85,B 0,C 180,E1 -7988.426,E2 -7988.426} C_VEL
LIN {X 0,Y 461.595,Z 631.977,A -85,B 0,C 180,E1 -7991.814,E2 -7991.814} C_VEL
LIN {X 0,Y 461.4,Z 638.573,A -85,B 0,C 180,E1 -7992.662,E2 -7992.662} C_VEL
LIN {X 0,Y 464.135,Z 666.427,A -85,B 0,C 180,E1 -7993.25,E2 -7993.25} C_VEL
LIN {X 0,Y 463.244,Z 750.603,A -85,B 0,C 180,E1 -7994.661,E2 -7994.661} C_VEL
LIN {X 0,Y 463.073,Z 764.389,A -85,B 0,C 180,E1 -7994.965,E2 -7994.965} C_VEL
LIN {X 0,Y 462.707,Z 776.092,A -85,B 0,C 180,E1 -7995.375,E2 -7995.375} C_VEL
LIN {X 0,Y 462.358,Z 787.371,A -85,B 0,C 180,E1 -7995.925,E2 -7995.925} C_VEL
LIN {X 0,Y 461.883,Z 799.391,A -85,B 0,C 180,E1 -7996.696,E2 -7996.696} C_VEL
LIN {X 0,Y 461.432,Z 809.695,A -85,B 0,C 180,E1 -7997.543,E2 -7997.543} C_VEL
LIN {X 0,Y 460.983,Z 819.754,A -85,B 0,C 180,E1 -7998.57,E2 -7998.57} C_VEL
LIN {X 0,Y 460.516,Z 828.578,A -85,B 0,C 180,E1 -7999.671,E2 -7999.671} C_VEL
LIN {X 0,Y 460.214,Z 835.842,A -85,B 0,C 180,E1 -8000.774,E2 -8000.774} C_VEL
LIN {X 0,Y 459.97,Z 842.957,A -85,B 0,C 180,E1 -8002.097,E2 -8002.097} C_VEL
LIN {X 0,Y 459.781,Z 848.888,A -85,B 0,C 180,E1 -8003.495,E2 -8003.495} C_VEL
LIN {X 0,Y 459.767,Z 853.032,A -85,B 0,C 180,E1 -8004.738,E2 -8004.738} C_VEL
LIN {X 0,Y 459.674,Z 855.361,A -85,B 0,C 180,E1 -8005.617,E2 -8005.617} C_VEL
LIN {X 0,Y 459.71,Z 857.26,A -85,B 0,C 180,E1 -8006.495,E2 -8006.495} C_VEL
LIN {X 0,Y 459.672,Z 858.692,A -85,B 0,C 180,E1 -8007.372,E2 -8007.372} C_VEL
LIN {X 0,Y 459.648,Z 860.318,A -85,B 0,C 180,E1 -8009.125,E2 -8009.125} C_VEL
LIN {X 0,Y 459.645,Z 860.538,A -85,B 0,C 180,E1 -8010.001,E2 -8010.001} C_VEL
LIN {X 0,Y 459.624,Z 860.316,A -85,B 0,C 180,E1 -8010.877,E2 -8010.877} C_VEL
LIN {X 0,Y 459.66,Z 858.688,A -85,B 0,C 180,E1 -8012.63,E2 -8012.63} C_VEL
LIN {X 0,Y 459.688,Z 857.255,A -85,B 0,C 180,E1 -8013.507,E2 -8013.507} C_VEL
LIN {X 0,Y 459.695,Z 854.27,A -85,B 0,C 180,E1 -8014.824,E2 -8014.824} C_VEL
LIN {X 0,Y 459.765,Z 850.217,A -85,B 0,C 180,E1 -8016.143,E2 -8016.143} C_VEL
LIN {X 0,Y 459.91,Z 843.956,A -85,B 0,C 180,E1 -8017.685,E2 -8017.685} C_VEL
LIN {X 0,Y 460.15,Z 837.123,A -85,B 0,C 180,E1 -8019.007,E2 -8019.007} C_VEL
LIN {X 0,Y 460.427,Z 830.137,A -85,B 0,C 180,E1 -8020.11,E2 -8020.11} C_VEL
LIN {X 0,Y 460.816,Z 821.691,A -85,B 0,C 180,E1 -8021.213,E2 -8021.213} C_VEL
LIN {X 0,Y 461.309,Z 811.209,A -85,B 0,C 180,E1 -8022.316,E2 -8022.316} C_VEL
LIN {X 0,Y 461.72,Z 800.804,A -85,B 0,C 180,E1 -8023.199,E2 -8023.199} C_VEL
LIN {X 0,Y 462.224,Z 789.314,A -85,B 0,C 180,E1 -8023.968,E2 -8023.968} C_VEL
LIN {X 0,Y 462.698,Z 777.34,A -85,B 0,C 180,E1 -8024.571,E2 -8024.571} C_VEL
LIN {X 0,Y 462.981,Z 765.225,A -85,B 0,C 180,E1 -8025.012,E2 -8025.012} C_VEL
LIN {X 0,Y 463.478,Z 747.168,A -85,B 0,C 180,E1 -8025.445,E2 -8025.445} C_VEL
LIN {X 0,Y 464.04,Z 665.209,A -85,B 0,C 180,E1 -8026.799,E2 -8026.799} C_VEL
LIN {X 0,Y 461.247,Z 642.132,A -85,B 0,C 180,E1 -8027.294,E2 -8027.294} C_VEL
LIN {X 0,Y 462.035,Z 620.745,A -85,B 0,C 180,E1 -8030.479,E2 -8030.479} C_VEL
LIN {X 0,Y 462.858,Z 600.711,A -85,B 0,C 180,E1 -8033.49,E2 -8033.49} C_VEL
LIN {X 0,Y 463.845,Z 579.274,A -85,B 0,C 180,E1 -8036.764,E2 -8036.764} C_VEL
LIN {X 0,Y 464.66,Z 563.609,A -85,B 0,C 180,E1 -8039.195,E2 -8039.195} C_VEL
LIN {X 0,Y 464.047,Z 558.816,A -85,B 0,C 180,E1 -8039.986,E2 -8039.986} C_VEL
LIN {X 0,Y 460.568,Z 543.118,A -85,B 0,C 180,E1 -8042.736,E2 -8042.736} C_VEL
LIN {X 0,Y 460.514,Z 543.122,A -85,B 0,C 180,E1 -8045.446,E2 -8045.446} C_VEL
LIN {X 0,Y 460.547,Z 543.12,A -85,B 0,C 180,E1 -8048.898,E2 -8048.898} C_VEL
LIN {X 0,Y 460.525,Z 543.117,A -85,B 0,C 180,E1 -8052.181,E2 -8052.181} C_VEL
LIN {X 0,Y 460.523,Z 543.121,A -85,B 0,C 180,E1 -8055.412,E2 -8055.412} C_VEL
LIN {X 0,Y 460.537,Z 543.11,A -85,B 0,C 180,E1 -8058.397,E2 -8058.397} C_VEL
LIN {X 0,Y 460.528,Z 543.121,A -85,B 0,C 180,E1 -8061.267,E2 -8061.267} C_VEL
LIN {X 0,Y 460.515,Z 543.114,A -85,B 0,C 180,E1 -8064.555,E2 -8064.555} C_VEL
LIN {X 0,Y 460.532,Z 543.112,A -85,B 0,C 180,E1 -8067.716,E2 -8067.716} C_VEL
LIN {X 0,Y 460.54,Z 543.113,A -85,B 0,C 180,E1 -8070.769,E2 -8070.769} C_VEL
LIN {X 0,Y 460.564,Z 543.109,A -85,B 0,C 180,E1 -8073.735,E2 -8073.735} C_VEL
LIN {X 0,Y 460.546,Z 543.108,A -85,B 0,C 180,E1 -8076.624,E2 -8076.624} C_VEL
LIN {X 0,Y 460.552,Z 543.118,A -85,B 0,C 180,E1 -8079.453,E2 -8079.453} C_VEL
LIN {X 0,Y 460.559,Z 543.101,A -85,B 0,C 180,E1 -8082.23,E2 -8082.23} C_VEL
LIN {X 0,Y 460.567,Z 543.111,A -85,B 0,C 180,E1 -8084.965,E2 -8084.965} C_VEL
LIN {X 0,Y 460.611,Z 543.098,A -85,B 0,C 180,E1 -8088.559,E2 -8088.559} C_VEL
LIN {X 0,Y 460.695,Z 543.096,A -85,B 0,C 180,E1 -8092.109,E2 -8092.109} C_VEL
LIN {X 0,Y 460.697,Z 543.093,A -85,B 0,C 180,E1 -8094.748,E2 -8094.748} C_VEL
LIN {X 0,Y 460.8,Z 543.074,A -85,B 0,C 180,E1 -8097.378,E2 -8097.378} C_VEL
LIN {X 0,Y 460.852,Z 543.079,A -85,B 0,C 180,E1 -8100,E2 -8100} C_VEL
LIN {X 0,Y 460.8,Z 543.079,A -85,B 0,C 180,E1 -8102.623,E2 -8102.623} C_VEL
LIN {X 0,Y 460.709,Z 543.092,A -85,B 0,C 180,E1 -8106.13,E2 -8106.13} C_VEL
LIN {X 0,Y 460.629,Z 543.103,A -85,B 0,C 180,E1 -8108.776,E2 -8108.776} C_VEL
LIN {X 0,Y 460.613,Z 543.096,A -85,B 0,C 180,E1 -8112.445,E2 -8112.445} C_VEL
LIN {X 0,Y 460.6,Z 543.113,A -85,B 0,C 180,E1 -8115.998,E2 -8115.998} C_VEL
LIN {X 0,Y 460.571,Z 543.101,A -85,B 0,C 180,E1 -8118.902,E2 -8118.902} C_VEL
LIN {X 0,Y 460.516,Z 543.117,A -85,B 0,C 180,E1 -8121.486,E2 -8121.486} C_VEL
LIN {X 0,Y 460.543,Z 543.11,A -85,B 0,C 180,E1 -8124.332,E2 -8124.332} C_VEL
LIN {X 0,Y 460.573,Z 543.109,A -85,B 0,C 180,E1 -8127.244,E2 -8127.244} C_VEL
LIN {X 0,Y 460.511,Z 543.117,A -85,B 0,C 180,E1 -8130.24,E2 -8130.24} C_VEL
LIN {X 0,Y 460.53,Z 543.117,A -85,B 0,C 180,E1 -8133.325,E2 -8133.325} C_VEL
LIN {X 0,Y 460.477,Z 543.127,A -85,B 0,C 180,E1 -8136.53,E2 -8136.53} C_VEL
LIN {X 0,Y 460.534,Z 543.117,A -85,B 0,C 180,E1 -8139.862,E2 -8139.862} C_VEL
LIN {X 0,Y 460.514,Z 543.115,A -85,B 0,C 180,E1 -8142.9,E2 -8142.9} C_VEL
LIN {X 0,Y 460.507,Z 543.121,A -85,B 0,C 180,E1 -8145.831,E2 -8145.831} C_VEL
LIN {X 0,Y 460.533,Z 543.117,A -85,B 0,C 180,E1 -8148.989,E2 -8148.989} C_VEL
LIN {X 0,Y 460.528,Z 543.113,A -85,B 0,C 180,E1 -8151.267,E2 -8151.267} C_VEL
LIN {X 0,Y 460.514,Z 543.123,A -85,B 0,C 180,E1 -8154.554,E2 -8154.554} C_VEL
LIN {X 0,Y 460.535,Z 543.119,A -85,B 0,C 180,E1 -8157.716,E2 -8157.716} C_VEL
LIN {X 0,Y 460.573,Z 543.173,A -85,B 0,C 180,E1 -8161.177,E2 -8161.177} C_VEL
LIN {X 0,Y 463.946,Z 558.176,A -85,B 0,C 180,E1 -8163.591,E2 -8163.591} C_VEL
LIN {X 0,Y 464.404,Z 562.193,A -85,B 0,C 180,E1 -8164.209,E2 -8164.209} C_VEL
LIN {X 0,Y 463.409,Z 584.514,A -85,B 0,C 180,E1 -8167.508,E2 -8167.508} C_VEL
LIN {X 0,Y 462.536,Z 608.237,A -85,B 0,C 180,E1 -8170.932,E2 -8170.932} C_VEL
LIN {X 0,Y 462.233,Z 622.068,A -85,B 0,C 180,E1 -8172.787,E2 -8172.787} C_VEL
LIN {X 0,Y 462.366,Z 622.872,A -85,B 0,C 180,E1 -8172.805,E2 -8172.805} C_VEL
LIN {X 0,Y 462.566,Z 628.712,A -85,B 0,C 180,E1 -8172.906,E2 -8172.906} C_VEL
LIN {X 0,Y 461.612,Z 634.576,A -85,B 0,C 180,E1 -8172.963,E2 -8172.963} C_VEL
LIN {X 0,Y 458.599,Z 646.257,A -85,B 0,C 180,E1 -8173.036,E2 -8173.036} C_VEL
LIN {X 0,Y 457.708,Z 652.191,A -85,B 0,C 180,E1 -8173.097,E2 -8173.097} C_VEL
LIN {X 0,Y 457.654,Z 654.182,A -85,B 0,C 180,E1 -8173.128,E2 -8173.128} C_VEL
LIN {X 0,Y 456.941,Z 732.35,A -85,B 0,C 180,E1 -8174.385,E2 -8174.385} C_VEL
LIN {X 0,Y 456.632,Z 745.7,A -85,B 0,C 180,E1 -8174.775,E2 -8174.775} C_VEL
LIN {X 0,Y 456.145,Z 758.212,A -85,B 0,C 180,E1 -8175.329,E2 -8175.329} C_VEL
LIN {X 0,Y 455.638,Z 770.298,A -85,B 0,C 180,E1 -8176.054,E2 -8176.054} C_VEL
LIN {X 0,Y 455.214,Z 780.631,A -85,B 0,C 180,E1 -8176.85,E2 -8176.85} C_VEL
LIN {X 0,Y 454.659,Z 790.959,A -85,B 0,C 180,E1 -8177.841,E2 -8177.841} C_VEL
LIN {X 0,Y 454.141,Z 799.544,A -85,B 0,C 180,E1 -8178.846,E2 -8178.846} C_VEL
LIN {X 0,Y 453.628,Z 808.878,A -85,B 0,C 180,E1 -8180.187,E2 -8180.187} C_VEL
LIN {X 0,Y 453.213,Z 816.305,A -85,B 0,C 180,E1 -8181.528,E2 -8181.528} C_VEL
LIN {X 0,Y 452.885,Z 822.272,A -85,B 0,C 180,E1 -8182.868,E2 -8182.868} C_VEL
LIN {X 0,Y 452.819,Z 826.987,A -85,B 0,C 180,E1 -8184.209,E2 -8184.209} C_VEL
LIN {X 0,Y 452.566,Z 830.6,A -85,B 0,C 180,E1 -8185.546,E2 -8185.546} C_VEL
LIN {X 0,Y 452.6,Z 832.457,A -85,B 0,C 180,E1 -8186.438,E2 -8186.438} C_VEL
LIN {X 0,Y 452.533,Z 833.881,A -85,B 0,C 180,E1 -8187.329,E2 -8187.329} C_VEL
LIN {X 0,Y 452.431,Z 835.495,A -85,B 0,C 180,E1 -8189.109,E2 -8189.109} C_VEL
LIN {X 0,Y 452.435,Z 835.732,A -85,B 0,C 180,E1 -8189.999,E2 -8189.999} C_VEL
LIN {X 0,Y 452.43,Z 835.544,A -85,B 0,C 180,E1 -8190.889,E2 -8190.889} C_VEL
LIN {X 0,Y 452.533,Z 833.995,A -85,B 0,C 180,E1 -8192.67,E2 -8192.67} C_VEL
LIN {X 0,Y 452.599,Z 832.635,A -85,B 0,C 180,E1 -8193.56,E2 -8193.56} C_VEL
LIN {X 0,Y 452.594,Z 829.774,A -85,B 0,C 180,E1 -8194.899,E2 -8194.899} C_VEL
LIN {X 0,Y 452.82,Z 825.88,A -85,B 0,C 180,E1 -8196.236,E2 -8196.236} C_VEL
LIN {X 0,Y 452.98,Z 820.844,A -85,B 0,C 180,E1 -8197.577,E2 -8197.577} C_VEL
LIN {X 0,Y 453.317,Z 814.492,A -85,B 0,C 180,E1 -8198.918,E2 -8198.918} C_VEL
LIN {X 0,Y 453.72,Z 806.592,A -85,B 0,C 180,E1 -8200.26,E2 -8200.26} C_VEL
LIN {X 0,Y 454.177,Z 798.517,A -85,B 0,C 180,E1 -8201.378,E2 -8201.378} C_VEL
LIN {X 0,Y 454.826,Z 788.615,A -85,B 0,C 180,E1 -8202.493,E2 -8202.493} C_VEL
LIN {X 0,Y 455.306,Z 777.757,A -85,B 0,C 180,E1 -8203.479,E2 -8203.479} C_VEL
LIN {X 0,Y 455.836,Z 766.616,A -85,B 0,C 180,E1 -8204.28,E2 -8204.28} C_VEL
LIN {X 0,Y 456.338,Z 754.426,A -85,B 0,C 180,E1 -8204.948,E2 -8204.948} C_VEL
LIN {X 0,Y 456.767,Z 740.978,A -85,B 0,C 180,E1 -8205.476,E2 -8205.476} C_VEL
LIN {X 0,Y 456.976,Z 728.701,A -85,B 0,C 180,E1 -8205.784,E2 -8205.784} C_VEL
LIN {X 0,Y 457.704,Z 638.817,A -85,B 0,C 180,E1 -8207.21,E2 -8207.21} C_VEL
LIN {X 0,Y 454.969,Z 622.713,A -85,B 0,C 180,E1 -8207.585,E2 -8207.585} C_VEL
LIN {X 0,Y 455.427,Z 606.571,A -85,B 0,C 180,E1 -8210.08,E2 -8210.08} C_VEL
LIN {X 0,Y 456.12,Z 587.873,A -85,B 0,C 180,E1 -8213.134,E2 -8213.134} C_VEL
LIN {X 0,Y 456.901,Z 570.733,A -85,B 0,C 180,E1 -8216,E2 -8216} C_VEL
LIN {X 0,Y 457.157,Z 561.992,A -85,B 0,C 180,E1 -8217.463,E2 -8217.463} C_VEL
LIN {X 0,Y 455.205,Z 551.457,A -85,B 0,C 180,E1 -8219.352,E2 -8219.352} C_VEL
LIN {X 0,Y 453.499,Z 543.999,A -85,B 0,C 180,E1 -8220.702,E2 -8220.702} C_VEL
LIN {X 0,Y 453.475,Z 543.999,A -85,B 0,C 180,E1 -8223.911,E2 -8223.911} C_VEL
LIN {X 0,Y 453.468,Z 544.003,A -85,B 0,C 180,E1 -8227.187,E2 -8227.187} C_VEL
LIN {X 0,Y 453.513,Z 543.99,A -85,B 0,C 180,E1 -8229.446,E2 -8229.446} C_VEL
LIN {X 0,Y 453.463,Z 543.993,A -85,B 0,C 180,E1 -8232.993,E2 -8232.993} C_VEL
LIN {X 0,Y 453.471,Z 543.998,A -85,B 0,C 180,E1 -8235.779,E2 -8235.779} C_VEL
LIN {X 0,Y 453.491,Z 543.994,A -85,B 0,C 180,E1 -8238.21,E2 -8238.21} C_VEL
LIN {X 0,Y 453.545,Z 543.992,A -85,B 0,C 180,E1 -8241.098,E2 -8241.098} C_VEL
LIN {X 0,Y 457.461,Z 555.551,A -85,B 0,C 180,E1 -8241.456,E2 -8241.456} C_VEL
LIN {X 0,Y 456.757,Z 623.704,A -85,B 0,C 180,E1 -8242.623,E2 -8242.623} C_VEL
LIN {X 0,Y 456.647,Z 637.027,A -85,B 0,C 180,E1 -8243.027,E2 -8243.027} C_VEL
LIN {X 0,Y 456.49,Z 649.417,A -85,B 0,C 180,E1 -8243.58,E2 -8243.58} C_VEL
LIN {X 0,Y 456.175,Z 660.987,A -85,B 0,C 180,E1 -8244.269,E2 -8244.269} C_VEL
LIN {X 0,Y 455.74,Z 673.15,A -85,B 0,C 180,E1 -8245.209,E2 -8245.209} C_VEL
LIN {X 0,Y 455.304,Z 683.772,A -85,B 0,C 180,E1 -8246.242,E2 -8246.242} C_VEL
LIN {X 0,Y 454.91,Z 692.34,A -85,B 0,C 180,E1 -8247.267,E2 -8247.267} C_VEL
LIN {X 0,Y 454.523,Z 701.039,A -85,B 0,C 180,E1 -8248.543,E2 -8248.543} C_VEL
LIN {X 0,Y 454.158,Z 707.714,A -85,B 0,C 180,E1 -8249.739,E2 -8249.739} C_VEL
LIN {X 0,Y 453.879,Z 713.705,A -85,B 0,C 180,E1 -8251.06,E2 -8251.06} C_VEL
LIN {X 0,Y 453.714,Z 718.214,A -85,B 0,C 180,E1 -8252.309,E2 -8252.309} C_VEL
LIN {X 0,Y 453.581,Z 721.111,A -85,B 0,C 180,E1 -8253.299,E2 -8253.299} C_VEL
LIN {X 0,Y 453.475,Z 723.391,A -85,B 0,C 180,E1 -8254.282,E2 -8254.282} C_VEL
LIN {X 0,Y 453.386,Z 725.175,A -85,B 0,C 180,E1 -8255.258,E2 -8255.258} C_VEL
LIN {X 0,Y 453.334,Z 726.401,A -85,B 0,C 180,E1 -8256.229,E2 -8256.229} C_VEL
LIN {X 0,Y 453.305,Z 727.173,A -85,B 0,C 180,E1 -8257.195,E2 -8257.195} C_VEL
LIN {X 0,Y 453.324,Z 727.445,A -85,B 0,C 180,E1 -8258.461,E2 -8258.461} C_VEL
LIN {X 0,Y 453.413,Z 726.649,A -85,B 0,C 180,E1 -8260.062,E2 -8260.062} C_VEL
LIN {X 0,Y 453.511,Z 725.543,A -85,B 0,C 180,E1 -8261.008,E2 -8261.008} C_VEL
LIN {X 0,Y 453.66,Z 723.024,A -85,B 0,C 180,E1 -8262.417,E2 -8262.417} C_VEL
LIN {X 0,Y 453.886,Z 719.402,A -85,B 0,C 180,E1 -8263.816,E2 -8263.816} C_VEL
LIN {X 0,Y 454.163,Z 714.603,A -85,B 0,C 180,E1 -8265.207,E2 -8265.207} C_VEL
LIN {X 0,Y 454.578,Z 708.463,A -85,B 0,C 180,E1 -8266.59,E2 -8266.59} C_VEL
LIN {X 0,Y 454.972,Z 700.785,A -85,B 0,C 180,E1 -8267.963,E2 -8267.963} C_VEL
LIN {X 0,Y 455.415,Z 692.854,A -85,B 0,C 180,E1 -8269.103,E2 -8269.103} C_VEL
LIN {X 0,Y 455.902,Z 683.161,A -85,B 0,C 180,E1 -8270.237,E2 -8270.237} C_VEL
LIN {X 0,Y 456.35,Z 672.354,A -85,B 0,C 180,E1 -8271.252,E2 -8271.252} C_VEL
LIN {X 0,Y 456.678,Z 661.801,A -85,B 0,C 180,E1 -8272.039,E2 -8272.039} C_VEL
LIN {X 0,Y 457.002,Z 649.135,A -85,B 0,C 180,E1 -8272.767,E2 -8272.767} C_VEL
LIN {X 0,Y 457.131,Z 636.424,A -85,B 0,C 180,E1 -8273.296,E2 -8273.296} C_VEL
LIN {X 0,Y 457.181,Z 622.896,A -85,B 0,C 180,E1 -8273.656,E2 -8273.656} C_VEL
LIN {X 0,Y 457.834,Z 555.311,A -85,B 0,C 180,E1 -8274.853,E2 -8274.853} C_VEL
LIN {X 0,Y 453.547,Z 543.99,A -85,B 0,C 180,E1 -8275.278,E2 -8275.278} C_VEL
LIN {X 0,Y 453.763,Z 543.962,A -85,B 0,C 180,E1 -8277.337,E2 -8277.337} C_VEL
LIN {X 0,Y 453.813,Z 543.957,A -85,B 0,C 180,E1 -8280,E2 -8280} C_VEL
LIN {X 0,Y 453.756,Z 543.968,A -85,B 0,C 180,E1 -8282.663,E2 -8282.663} C_VEL
LIN {X 0,Y 453.674,Z 543.973,A -85,B 0,C 180,E1 -8286.225,E2 -8286.225} C_VEL
LIN {X 0,Y 453.583,Z 543.986,A -85,B 0,C 180,E1 -8288.914,E2 -8288.914} C_VEL
LIN {X 0,Y 453.59,Z 543.983,A -85,B 0,C 180,E1 -8292.551,E2 -8292.551} C_VEL
LIN {X 0,Y 453.534,Z 543.985,A -85,B 0,C 180,E1 -8296.196,E2 -8296.196} C_VEL
LIN {X 0,Y 453.51,Z 543.994,A -85,B 0,C 180,E1 -8299.041,E2 -8299.041} C_VEL
LIN {X 0,Y 453.466,Z 543.996,A -85,B 0,C 180,E1 -8301.837,E2 -8301.837} C_VEL
LIN {X 0,Y 453.504,Z 543.996,A -85,B 0,C 180,E1 -8304.735,E2 -8304.735} C_VEL
LIN {X 0,Y 453.529,Z 543.987,A -85,B 0,C 180,E1 -8307.962,E2 -8307.962} C_VEL
LIN {X 0,Y 453.474,Z 544,A -85,B 0,C 180,E1 -8310.76,E2 -8310.76} C_VEL
LIN {X 0,Y 453.47,Z 543.996,A -85,B 0,C 180,E1 -8313.913,E2 -8313.913} C_VEL
LIN {X 0,Y 453.464,Z 543.997,A -85,B 0,C 180,E1 -8317.189,E2 -8317.189} C_VEL
LIN {X 0,Y 453.526,Z 543.99,A -85,B 0,C 180,E1 -8319.446,E2 -8319.446} C_VEL
LIN {X 0,Y 453.486,Z 543.998,A -85,B 0,C 180,E1 -8322.992,E2 -8322.992} C_VEL
LIN {X 0,Y 453.471,Z 543.998,A -85,B 0,C 180,E1 -8325.782,E2 -8325.782} C_VEL
LIN {X 0,Y 453.491,Z 543.996,A -85,B 0,C 180,E1 -8328.212,E2 -8328.212} C_VEL
LIN {X 0,Y 453.528,Z 543.993,A -85,B 0,C 180,E1 -8330.788,E2 -8330.788} C_VEL
LIN {X 0,Y 453.454,Z 544.002,A -85,B 0,C 180,E1 -8333.919,E2 -8333.919} C_VEL
LIN {X 0,Y 453.48,Z 544.001,A -85,B 0,C 180,E1 -8337.152,E2 -8337.152} C_VEL
LIN {X 0,Y 453.519,Z 544.022,A -85,B 0,C 180,E1 -8339,E2 -8339} C_VEL
LIN {X 0,Y 456.693,Z 557.892,A -85,B 0,C 180,E1 -8341.303,E2 -8341.303} C_VEL
LIN {X 0,Y 457.584,Z 562.715,A -85,B 0,C 180,E1 -8342.068,E2 -8342.068} C_VEL
LIN {X 0,Y 456.776,Z 579.676,A -85,B 0,C 180,E1 -8344.482,E2 -8344.482} C_VEL
LIN {X 0,Y 455.592,Z 605,A -85,B 0,C 180,E1 -8348.002,E2 -8348.002} C_VEL
LIN {X 0,Y 454.608,Z 630.917,A -85,B 0,C 180,E1 -8351.524,E2 -8351.524} C_VEL
LIN {X 0,Y 454.391,Z 637.447,A -85,B 0,C 180,E1 -8352.366,E2 -8352.366} C_VEL
LIN {X 0,Y 457.333,Z 666.326,A -85,B 0,C 180,E1 -8352.999,E2 -8352.999} C_VEL
LIN {X 0,Y 456.362,Z 757.794,A -85,B 0,C 180,E1 -8354.567,E2 -8354.567} C_VEL
LIN {X 0,Y 455.988,Z 771.014,A -85,B 0,C 180,E1 -8354.954,E2 -8354.954} C_VEL
LIN {X 0,Y 455.54,Z 784.218,A -85,B 0,C 180,E1 -8355.539,E2 -8355.539} C_VEL
LIN {X 0,Y 455.102,Z 796.075,A -85,B 0,C 180,E1 -8356.266,E2 -8356.266} C_VEL
LIN {X 0,Y 454.569,Z 807.349,A -85,B 0,C 180,E1 -8357.154,E2 -8357.154} C_VEL
LIN {X 0,Y 454.026,Z 817.618,A -85,B 0,C 180,E1 -8358.166,E2 -8358.166} C_VEL
LIN {X 0,Y 453.558,Z 826.763,A -85,B 0,C 180,E1 -8359.285,E2 -8359.285} C_VEL
LIN {X 0,Y 453.181,Z 835.656,A -85,B 0,C 180,E1 -8360.629,E2 -8360.629} C_VEL
LIN {X 0,Y 452.906,Z 842.768,A -85,B 0,C 180,E1 -8361.973,E2 -8361.973} C_VEL
LIN {X 0,Y 452.69,Z 849.14,A -85,B 0,C 180,E1 -8363.515,E2 -8363.515} C_VEL
LIN {X 0,Y 452.632,Z 854.085,A -85,B 0,C 180,E1 -8365.102,E2 -8365.102} C_VEL
LIN {X 0,Y 452.605,Z 857.068,A -85,B 0,C 180,E1 -8366.44,E2 -8366.44} C_VEL
LIN {X 0,Y 452.593,Z 858.5,A -85,B 0,C 180,E1 -8367.331,E2 -8367.331} C_VEL
LIN {X 0,Y 452.577,Z 860.125,A -85,B 0,C 180,E1 -8369.111,E2 -8369.111} C_VEL
LIN {X 0,Y 452.572,Z 860.346,A -85,B 0,C 180,E1 -8370.001,E2 -8370.001} C_VEL
LIN {X 0,Y 452.538,Z 859.505,A -85,B 0,C 180,E1 -8371.781,E2 -8371.781} C_VEL
LIN {X 0,Y 452.581,Z 858.496,A -85,B 0,C 180,E1 -8372.671,E2 -8372.671} C_VEL
LIN {X 0,Y 452.584,Z 857.062,A -85,B 0,C 180,E1 -8373.562,E2 -8373.562} C_VEL
LIN {X 0,Y 452.622,Z 854.078,A -85,B 0,C 180,E1 -8374.9,E2 -8374.9} C_VEL
LIN {X 0,Y 452.732,Z 848.969,A -85,B 0,C 180,E1 -8376.531,E2 -8376.531} C_VEL
LIN {X 0,Y 452.895,Z 842.754,A -85,B 0,C 180,E1 -8378.029,E2 -8378.029} C_VEL
LIN {X 0,Y 453.181,Z 835.635,A -85,B 0,C 180,E1 -8379.372,E2 -8379.372} C_VEL
LIN {X 0,Y 453.537,Z 826.751,A -85,B 0,C 180,E1 -8380.717,E2 -8380.717} C_VEL
LIN {X 0,Y 454.013,Z 817.606,A -85,B 0,C 180,E1 -8381.836,E2 -8381.836} C_VEL
LIN {X 0,Y 454.577,Z 806.731,A -85,B 0,C 180,E1 -8382.9,E2 -8382.9} C_VEL
LIN {X 0,Y 455.041,Z 796.039,A -85,B 0,C 180,E1 -8383.737,E2 -8383.737} C_VEL
LIN {X 0,Y 455.544,Z 784.173,A -85,B 0,C 180,E1 -8384.462,E2 -8384.462} C_VEL
LIN {X 0,Y 455.928,Z 771.701,A -85,B 0,C 180,E1 -8385.021,E2 -8385.021} C_VEL
LIN {X 0,Y 456.325,Z 758.83,A -85,B 0,C 180,E1 -8385.407,E2 -8385.407} C_VEL
LIN {X 0,Y 456.663,Z 735.055,A -85,B 0,C 180,E1 -8385.854,E2 -8385.854} C_VEL
LIN {X 0,Y 457.298,Z 666.745,A -85,B 0,C 180,E1 -8387.001,E2 -8387.001} C_VEL
LIN {X 0,Y 454.219,Z 641.212,A -85,B 0,C 180,E1 -8387.568,E2 -8387.568} C_VEL
LIN {X 0,Y 455.014,Z 621.326,A -85,B 0,C 180,E1 -8390.573,E2 -8390.573} C_VEL
LIN {X 0,Y 455.884,Z 601.354,A -85,B 0,C 180,E1 -8393.63,E2 -8393.63} C_VEL
LIN {X 0,Y 456.901,Z 580.59,A -85,B 0,C 180,E1 -8396.855,E2 -8396.855} C_VEL
LIN {X 0,Y 457.758,Z 564.251,A -85,B 0,C 180,E1 -8399.426,E2 -8399.426} C_VEL
LIN {X 0,Y 455.907,Z 554.598,A -85,B 0,C 180,E1 -8401.092,E2 -8401.092} C_VEL
LIN {X 0,Y 453.509,Z 543.997,A -85,B 0,C 180,E1 -8403.017,E2 -8403.017} C_VEL
LIN {X 0,Y 453.456,Z 544,A -85,B 0,C 180,E1 -8406.299,E2 -8406.299} C_VEL
LIN {X 0,Y 453.507,Z 543.994,A -85,B 0,C 180,E1 -8409.448,E2 -8409.448} C_VEL
LIN {X 0,Y 453.466,Z 544,A -85,B 0,C 180,E1 -8412.995,E2 -8412.995} C_VEL
LIN {X 0,Y 453.478,Z 543.995,A -85,B 0,C 180,E1 -8415.78,E2 -8415.78} C_VEL
LIN {X 0,Y 453.496,Z 543.996,A -85,B 0,C 180,E1 -8419.391,E2 -8419.391} C_VEL
LIN {X 0,Y 453.474,Z 543.992,A -85,B 0,C 180,E1 -8422.223,E2 -8422.223} C_VEL
LIN {X 0,Y 453.49,Z 543.997,A -85,B 0,C 180,E1 -8425.222,E2 -8425.222} C_VEL
LIN {X 0,Y 453.466,Z 543.99,A -85,B 0,C 180,E1 -8428.475,E2 -8428.475} C_VEL
LIN {X 0,Y 453.533,Z 543.988,A -85,B 0,C 180,E1 -8432.04,E2 -8432.04} C_VEL
LIN {X 0,Y 453.514,Z 543.985,A -85,B 0,C 180,E1 -8435.266,E2 -8435.266} C_VEL
LIN {X 0,Y 453.48,Z 543.993,A -85,B 0,C 180,E1 -8438.415,E2 -8438.415} C_VEL
LIN {X 0,Y 453.522,Z 543.988,A -85,B 0,C 180,E1 -8441.009,E2 -8441.009} C_VEL
LIN {X 0,Y 453.569,Z 543.984,A -85,B 0,C 180,E1 -8443.88,E2 -8443.88} C_VEL
LIN {X 0,Y 453.563,Z 543.985,A -85,B 0,C 180,E1 -8447.471,E2 -8447.471} C_VEL
LIN {X 0,Y 453.592,Z 543.974,A -85,B 0,C 180,E1 -8451.087,E2 -8451.087} C_VEL
LIN {X 0,Y 453.677,Z 543.974,A -85,B 0,C 180,E1 -8453.775,E2 -8453.775} C_VEL
LIN {X 0,Y 453.744,Z 543.953,A -85,B 0,C 180,E1 -8457.337,E2 -8457.337} C_VEL
LIN {X 0,Y 453.822,Z 543.955,A -85,B 0,C 180,E1 -8460,E2 -8460} C_VEL
LIN {X 0,Y 453.745,Z 543.958,A -85,B 0,C 180,E1 -8462.663,E2 -8462.663} C_VEL
LIN {X 0,Y 453.677,Z 543.967,A -85,B 0,C 180,E1 -8466.225,E2 -8466.225} C_VEL
LIN {X 0,Y 453.592,Z 543.98,A -85,B 0,C 180,E1 -8468.913,E2 -8468.913} C_VEL
LIN {X 0,Y 453.564,Z 543.974,A -85,B 0,C 180,E1 -8472.529,E2 -8472.529} C_VEL
LIN {X 0,Y 453.545,Z 543.989,A -85,B 0,C 180,E1 -8476.196,E2 -8476.196} C_VEL
LIN {X 0,Y 453.52,Z 543.979,A -85,B 0,C 180,E1 -8479.041,E2 -8479.041} C_VEL
LIN {X 0,Y 453.477,Z 543.998,A -85,B 0,C 180,E1 -8481.836,E2 -8481.836} C_VEL
LIN {X 0,Y 453.515,Z 543.982,A -85,B 0,C 180,E1 -8484.735,E2 -8484.735} C_VEL
LIN {X 0,Y 453.533,Z 543.993,A -85,B 0,C 180,E1 -8487.96,E2 -8487.96} C_VEL
LIN {X 0,Y 453.466,Z 543.992,A -85,B 0,C 180,E1 -8491.525,E2 -8491.525} C_VEL
LIN {X 0,Y 453.488,Z 543.99,A -85,B 0,C 180,E1 -8494.777,E2 -8494.777} C_VEL
LIN {X 0,Y 453.466,Z 544.001,A -85,B 0,C 180,E1 -8498.312,E2 -8498.312} C_VEL
LIN {X 0,Y 453.496,Z 543.996,A -85,B 0,C 180,E1 -8500.609,E2 -8500.609} C_VEL
LIN {X 0,Y 453.456,Z 543.993,A -85,B 0,C 180,E1 -8503.244,E2 -8503.244} C_VEL
LIN {X 0,Y 453.462,Z 543.999,A -85,B 0,C 180,E1 -8505.778,E2 -8505.778} C_VEL
LIN {X 0,Y 453.497,Z 543.993,A -85,B 0,C 180,E1 -8509.409,E2 -8509.409} C_VEL
LIN {X 0,Y 453.452,Z 543.995,A -85,B 0,C 180,E1 -8512.227,E2 -8512.227} C_VEL
LIN {X 0,Y 453.491,Z 543.995,A -85,B 0,C 180,E1 -8515.223,E2 -8515.223} C_VEL
LIN {X 0,Y 453.47,Z 544.001,A -85,B 0,C 180,E1 -8518.475,E2 -8518.475} C_VEL
LIN {X 0,Y 453.541,Z 544.081,A -85,B 0,C 180,E1 -8520.91,E2 -8520.91} C_VEL
LIN {X 0,Y 457.146,Z 560.145,A -85,B 0,C 180,E1 -8523.523,E2 -8523.523} C_VEL
LIN {X 0,Y 457.508,Z 565.068,A -85,B 0,C 180,E1 -8524.28,E2 -8524.28} C_VEL
LIN {X 0,Y 456.406,Z 587.579,A -85,B 0,C 180,E1 -8527.634,E2 -8527.634} C_VEL
LIN {X 0,Y 455.618,Z 609.969,A -85,B 0,C 180,E1 -8530.875,E2 -8530.875} C_VEL
LIN {X 0,Y 455.284,Z 621.905,A -85,B 0,C 180,E1 -8532.508,E2 -8532.508} C_VEL
LIN {X 0,Y 457.765,Z 637.57,A -85,B 0,C 180,E1 -8532.863,E2 -8532.863} C_VEL
LIN {X 0,Y 457.654,Z 654.182,A -85,B 0,C 180,E1 -8533.128,E2 -8533.128} C_VEL
LIN {X 0,Y 457.047,Z 660.028,A -85,B 0,C 180,E1 -8533.199,E2 -8533.199} C_VEL
LIN {X 0,Y 451.36,Z 679.04,A -85,B 0,C 180,E1 -8533.291,E2 -8533.291} C_VEL
LIN {X 0,Y 450.667,Z 684.89,A -85,B 0,C 180,E1 -8533.36,E2 -8533.36} C_VEL
LIN {X 0,Y 450.132,Z 732.466,A -85,B 0,C 180,E1 -8534.143,E2 -8534.143} C_VEL
LIN {X 0,Y 449.811,Z 745.853,A -85,B 0,C 180,E1 -8534.538,E2 -8534.538} C_VEL
LIN {X 0,Y 449.282,Z 758.381,A -85,B 0,C 180,E1 -8535.1,E2 -8535.1} C_VEL
LIN {X 0,Y 448.745,Z 770.476,A -85,B 0,C 180,E1 -8535.835,E2 -8535.835} C_VEL
LIN {X 0,Y 448.25,Z 781.913,A -85,B 0,C 180,E1 -8536.743,E2 -8536.743} C_VEL
LIN {X 0,Y 447.589,Z 793.211,A -85,B 0,C 180,E1 -8537.876,E2 -8537.876} C_VEL
LIN {X 0,Y 447.086,Z 801.458,A -85,B 0,C 180,E1 -8538.897,E2 -8538.897} C_VEL
LIN {X 0,Y 446.527,Z 810.399,A -85,B 0,C 180,E1 -8540.258,E2 -8540.258} C_VEL
LIN {X 0,Y 446.103,Z 817.584,A -85,B 0,C 180,E1 -8541.62,E2 -8541.62} C_VEL
LIN {X 0,Y 445.801,Z 823.57,A -85,B 0,C 180,E1 -8543.039,E2 -8543.039} C_VEL
LIN {X 0,Y 445.647,Z 828.513,A -85,B 0,C 180,E1 -8544.57,E2 -8544.57} C_VEL
LIN {X 0,Y 445.485,Z 830.793,A -85,B 0,C 180,E1 -8545.475,E2 -8545.475} C_VEL
LIN {X 0,Y 445.502,Z 832.65,A -85,B 0,C 180,E1 -8546.381,E2 -8546.381} C_VEL
LIN {X 0,Y 445.462,Z 834.074,A -85,B 0,C 180,E1 -8547.286,E2 -8547.286} C_VEL
LIN {X 0,Y 445.341,Z 835.688,A -85,B 0,C 180,E1 -8549.095,E2 -8549.095} C_VEL
LIN {X 0,Y 445.342,Z 835.925,A -85,B 0,C 180,E1 -8549.999,E2 -8549.999} C_VEL
LIN {X 0,Y 445.341,Z 835.736,A -85,B 0,C 180,E1 -8550.903,E2 -8550.903} C_VEL
LIN {X 0,Y 445.462,Z 834.187,A -85,B 0,C 180,E1 -8552.712,E2 -8552.712} C_VEL
LIN {X 0,Y 445.501,Z 832.827,A -85,B 0,C 180,E1 -8553.617,E2 -8553.617} C_VEL
LIN {X 0,Y 445.532,Z 829.964,A -85,B 0,C 180,E1 -8554.976,E2 -8554.976} C_VEL
LIN {X 0,Y 445.757,Z 826.069,A -85,B 0,C 180,E1 -8556.335,E2 -8556.335} C_VEL
LIN {X 0,Y 445.933,Z 821.032,A -85,B 0,C 180,E1 -8557.698,E2 -8557.698} C_VEL
LIN {X 0,Y 446.282,Z 814.679,A -85,B 0,C 180,E1 -8559.06,E2 -8559.06} C_VEL
LIN {X 0,Y 446.742,Z 806.775,A -85,B 0,C 180,E1 -8560.422,E2 -8560.422} C_VEL
LIN {X 0,Y 447.225,Z 798.697,A -85,B 0,C 180,E1 -8561.557,E2 -8561.557} C_VEL
LIN {X 0,Y 447.896,Z 788.79,A -85,B 0,C 180,E1 -8562.689,E2 -8562.689} C_VEL
LIN {X 0,Y 448.383,Z 778.534,A -85,B 0,C 180,E1 -8563.639,E2 -8563.639} C_VEL
LIN {X 0,Y 448.965,Z 766.777,A -85,B 0,C 180,E1 -8564.504,E2 -8564.504} C_VEL
LIN {X 0,Y 449.487,Z 754.571,A -85,B 0,C 180,E1 -8565.182,E2 -8565.182} C_VEL
LIN {X 0,Y 449.928,Z 741.097,A -85,B 0,C 180,E1 -8565.718,E2 -8565.718} C_VEL
LIN {X 0,Y 450.158,Z 728.746,A -85,B 0,C 180,E1 -8566.029,E2 -8566.029} C_VEL
LIN {X 0,Y 450.933,Z 639.687,A -85,B 0,C 180,E1 -8567.463,E2 -8567.463} C_VEL
LIN {X 0,Y 448.072,Z 622.774,A -85,B 0,C 180,E1 -8567.873,E2 -8567.873} C_VEL
LIN {X 0,Y 448.55,Z 606.539,A -85,B 0,C 180,E1 -8570.402,E2 -8570.402} C_VEL
LIN {X 0,Y 449.339,Z 587.694,A -85,B 0,C 180,E1 -8573.504,E2 -8573.504} C_VEL
LIN {X 0,Y 450.06,Z 570.398,A -85,B 0,C 180,E1 -8576.425,E2 -8576.425} C_VEL
LIN {X 0,Y 450.265,Z 563.027,A -85,B 0,C 180,E1 -8577.672,E2 -8577.672} C_VEL
LIN {X 0,Y 448.206,Z 552.456,A -85,B 0,C 180,E1 -8579.598,E2 -8579.598} C_VEL
LIN {X 0,Y 446.461,Z 544.874,A -85,B 0,C 180,E1 -8580.999,E2 -8580.999} C_VEL
LIN {X 0,Y 446.428,Z 544.878,A -85,B 0,C 180,E1 -8584.522,E2 -8584.522} C_VEL
LIN {X 0,Y 446.427,Z 544.877,A -85,B 0,C 180,E1 -8588.081,E2 -8588.081} C_VEL
LIN {X 0,Y 446.423,Z 544.876,A -85,B 0,C 180,E1 -8590.917,E2 -8590.917} C_VEL
LIN {X 0,Y 446.418,Z 544.868,A -85,B 0,C 180,E1 -8593.842,E2 -8593.842} C_VEL
LIN {X 0,Y 446.441,Z 544.871,A -85,B 0,C 180,E1 -8596.396,E2 -8596.396} C_VEL
LIN {X 0,Y 446.464,Z 544.873,A -85,B 0,C 180,E1 -8599.804,E2 -8599.804} C_VEL
LIN {X 0,Y 446.531,Z 545.066,A -85,B 0,C 180,E1 -8600.868,E2 -8600.868} C_VEL
LIN {X 0,Y 450.605,Z 557.394,A -85,B 0,C 180,E1 -8601.244,E2 -8601.244} C_VEL
LIN {X 0,Y 449.885,Z 625.077,A -85,B 0,C 180,E1 -8602.433,E2 -8602.433} C_VEL
LIN {X 0,Y 449.773,Z 638.761,A -85,B 0,C 180,E1 -8602.864,E2 -8602.864} C_VEL
LIN {X 0,Y 449.556,Z 651.189,A -85,B 0,C 180,E1 -8603.436,E2 -8603.436} C_VEL
LIN {X 0,Y 449.23,Z 663.264,A -85,B 0,C 180,E1 -8604.189,E2 -8604.189} C_VEL
LIN {X 0,Y 448.793,Z 675.145,A -85,B 0,C 180,E1 -8605.139,E2 -8605.139} C_VEL
LIN {X 0,Y 448.329,Z 685.483,A -85,B 0,C 180,E1 -8606.181,E2 -8606.181} C_VEL
LIN {X 0,Y 447.829,Z 695.848,A -85,B 0,C 180,E1 -8607.486,E2 -8607.486} C_VEL
LIN {X 0,Y 447.457,Z 704.101,A -85,B 0,C 180,E1 -8608.78,E2 -8608.78} C_VEL
LIN {X 0,Y 447.045,Z 711.896,A -85,B 0,C 180,E1 -8610.323,E2 -8610.323} C_VEL
LIN {X 0,Y 446.745,Z 717.879,A -85,B 0,C 180,E1 -8611.839,E2 -8611.839} C_VEL
LIN {X 0,Y 446.553,Z 722.342,A -85,B 0,C 180,E1 -8613.35,E2 -8613.35} C_VEL
LIN {X 0,Y 446.402,Z 725.508,A -85,B 0,C 180,E1 -8614.844,E2 -8614.844} C_VEL
LIN {X 0,Y 446.309,Z 727.153,A -85,B 0,C 180,E1 -8615.965,E2 -8615.965} C_VEL
LIN {X 0,Y 446.302,Z 727.939,A -85,B 0,C 180,E1 -8616.816,E2 -8616.816} C_VEL
LIN {X 0,Y 446.321,Z 728.482,A -85,B 0,C 180,E1 -8618.282,E2 -8618.282} C_VEL
LIN {X 0,Y 446.381,Z 727.976,A -85,B 0,C 180,E1 -8619.734,E2 -8619.734} C_VEL
LIN {X 0,Y 446.49,Z 726.939,A -85,B 0,C 180,E1 -8620.805,E2 -8620.805} C_VEL
LIN {X 0,Y 446.565,Z 725.711,A -85,B 0,C 180,E1 -8621.654,E2 -8621.654} C_VEL
LIN {X 0,Y 446.794,Z 722.745,A -85,B 0,C 180,E1 -8623.082,E2 -8623.082} C_VEL
LIN {X 0,Y 447.053,Z 718.651,A -85,B 0,C 180,E1 -8624.499,E2 -8624.499} C_VEL
LIN {X 0,Y 447.388,Z 713.321,A -85,B 0,C 180,E1 -8625.907,E2 -8625.907} C_VEL
LIN {X 0,Y 447.81,Z 706.583,A -85,B 0,C 180,E1 -8627.307,E2 -8627.307} C_VEL
LIN {X 0,Y 448.213,Z 699.676,A -85,B 0,C 180,E1 -8628.468,E2 -8628.468} C_VEL
LIN {X 0,Y 448.696,Z 691.307,A -85,B 0,C 180,E1 -8629.623,E2 -8629.623} C_VEL
LIN {X 0,Y 449.125,Z 681.962,A -85,B 0,C 180,E1 -8630.674,E2 -8630.674} C_VEL
LIN {X 0,Y 449.633,Z 670.738,A -85,B 0,C 180,E1 -8631.687,E2 -8631.687} C_VEL
LIN {X 0,Y 450.047,Z 659.518,A -85,B 0,C 180,E1 -8632.485,E2 -8632.485} C_VEL
LIN {X 0,Y 450.291,Z 646.878,A -85,B 0,C 180,E1 -8633.165,E2 -8633.165} C_VEL
LIN {X 0,Y 450.421,Z 633.594,A -85,B 0,C 180,E1 -8633.673,E2 -8633.673} C_VEL
LIN {X 0,Y 450.427,Z 620.322,A -85,B 0,C 180,E1 -8633.982,E2 -8633.982} C_VEL
LIN {X 0,Y 451.094,Z 556.744,A -85,B 0,C 180,E1 -8635.132,E2 -8635.132} C_VEL
LIN {X 0,Y 446.508,Z 545.185,A -85,B 0,C 180,E1 -8635.571,E2 -8635.571} C_VEL
LIN {X 0,Y 446.486,Z 544.869,A -85,B 0,C 180,E1 -8635.599,E2 -8635.599} C_VEL
LIN {X 0,Y 446.708,Z 544.841,A -85,B 0,C 180,E1 -8637.295,E2 -8637.295} C_VEL
LIN {X 0,Y 446.784,Z 544.833,A -85,B 0,C 180,E1 -8640,E2 -8640} C_VEL
LIN {X 0,Y 446.7,Z 544.846,A -85,B 0,C 180,E1 -8642.705,E2 -8642.705} C_VEL
LIN {X 0,Y 446.641,Z 544.85,A -85,B 0,C 180,E1 -8646.324,E2 -8646.324} C_VEL
LIN {X 0,Y 446.529,Z 544.863,A -85,B 0,C 180,E1 -8649.056,E2 -8649.056} C_VEL
LIN {X 0,Y 446.523,Z 544.863,A -85,B 0,C 180,E1 -8652.73,E2 -8652.73} C_VEL
LIN {X 0,Y 446.479,Z 544.866,A -85,B 0,C 180,E1 -8656.459,E2 -8656.459} C_VEL
LIN {X 0,Y 446.459,Z 544.87,A -85,B 0,C 180,E1 -8659.304,E2 -8659.304} C_VEL
LIN {X 0,Y 446.408,Z 544.877,A -85,B 0,C 180,E1 -8662.2,E2 -8662.2} C_VEL
LIN {X 0,Y 446.448,Z 544.873,A -85,B 0,C 180,E1 -8665.153,E2 -8665.153} C_VEL
LIN {X 0,Y 446.475,Z 544.867,A -85,B 0,C 180,E1 -8668.179,E2 -8668.179} C_VEL
LIN {X 0,Y 446.411,Z 544.878,A -85,B 0,C 180,E1 -8671.301,E2 -8671.301} C_VEL
LIN {X 0,Y 446.422,Z 544.875,A -85,B 0,C 180,E1 -8674.524,E2 -8674.524} C_VEL
LIN {X 0,Y 446.431,Z 544.871,A -85,B 0,C 180,E1 -8678.084,E2 -8678.084} C_VEL
LIN {X 0,Y 446.441,Z 544.876,A -85,B 0,C 180,E1 -8680.922,E2 -8680.922} C_VEL
LIN {X 0,Y 446.439,Z 544.874,A -85,B 0,C 180,E1 -8683.841,E2 -8683.841} C_VEL
LIN {X 0,Y 446.441,Z 544.876,A -85,B 0,C 180,E1 -8686.398,E2 -8686.398} C_VEL
LIN {X 0,Y 446.464,Z 544.87,A -85,B 0,C 180,E1 -8689.806,E2 -8689.806} C_VEL
LIN {X 0,Y 446.431,Z 544.875,A -85,B 0,C 180,E1 -8692.125,E2 -8692.125} C_VEL
LIN {X 0,Y 446.427,Z 544.878,A -85,B 0,C 180,E1 -8695.478,E2 -8695.478} C_VEL
LIN {X 0,Y 446.458,Z 544.971,A -85,B 0,C 180,E1 -8698.683,E2 -8698.683} C_VEL
LIN {X 0,Y 449.723,Z 558.877,A -85,B 0,C 180,E1 -8701.061,E2 -8701.061} C_VEL
LIN {X 0,Y 450.765,Z 565.463,A -85,B 0,C 180,E1 -8702.114,E2 -8702.114} C_VEL
LIN {X 0,Y 449.573,Z 585.775,A -85,B 0,C 180,E1 -8705.053,E2 -8705.053} C_VEL
LIN {X 0,Y 448.422,Z 609.438,A -85,B 0,C 180,E1 -8708.39,E2 -8708.39} C_VEL
LIN {X 0,Y 447.568,Z 631.66,A -85,B 0,C 180,E1 -8711.46,E2 -8711.46} C_VEL
LIN {X 0,Y 447.406,Z 636.003,A -85,B 0,C 180,E1 -8712.049,E2 -8712.049} C_VEL
LIN {X 0,Y 450.546,Z 667.574,A -85,B 0,C 180,E1 -8712.761,E2 -8712.761} C_VEL
LIN {X 0,Y 449.505,Z 758.837,A -85,B 0,C 180,E1 -8714.354,E2 -8714.354} C_VEL
LIN {X 0,Y 449.119,Z 771.632,A -85,B 0,C 180,E1 -8714.748,E2 -8714.748} C_VEL
LIN {X 0,Y 448.657,Z 784.061,A -85,B 0,C 180,E1 -8715.312,E2 -8715.312} C_VEL
LIN {X 0,Y 448.179,Z 795.906,A -85,B 0,C 180,E1 -8716.05,E2 -8716.05} C_VEL
LIN {X 0,Y 447.653,Z 807.057,A -85,B 0,C 180,E1 -8716.941,E2 -8716.941} C_VEL
LIN {X 0,Y 447.073,Z 817.437,A -85,B 0,C 180,E1 -8717.979,E2 -8717.979} C_VEL
LIN {X 0,Y 446.548,Z 826.579,A -85,B 0,C 180,E1 -8719.115,E2 -8719.115} C_VEL
LIN {X 0,Y 446.13,Z 835.468,A -85,B 0,C 180,E1 -8720.48,E2 -8720.48} C_VEL
LIN {X 0,Y 445.857,Z 842.58,A -85,B 0,C 180,E1 -8721.845,E2 -8721.845} C_VEL
LIN {X 0,Y 445.655,Z 848.386,A -85,B 0,C 180,E1 -8723.254,E2 -8723.254} C_VEL
LIN {X 0,Y 445.586,Z 852.65,A -85,B 0,C 180,E1 -8724.571,E2 -8724.571} C_VEL
LIN {X 0,Y 445.508,Z 854.978,A -85,B 0,C 180,E1 -8725.477,E2 -8725.477} C_VEL
LIN {X 0,Y 445.501,Z 856.875,A -85,B 0,C 180,E1 -8726.383,E2 -8726.383} C_VEL
LIN {X 0,Y 445.516,Z 858.308,A -85,B 0,C 180,E1 -8727.288,E2 -8727.288} C_VEL
LIN {X 0,Y 445.479,Z 859.932,A -85,B 0,C 180,E1 -8729.097,E2 -8729.097} C_VEL
LIN {X 0,Y 445.501,Z 860.154,A -85,B 0,C 180,E1 -8730.001,E2 -8730.001} C_VEL
LIN {X 0,Y 445.451,Z 859.312,A -85,B 0,C 180,E1 -8731.809,E2 -8731.809} C_VEL
LIN {X 0,Y 445.504,Z 858.303,A -85,B 0,C 180,E1 -8732.713,E2 -8732.713} C_VEL
LIN {X 0,Y 445.481,Z 856.869,A -85,B 0,C 180,E1 -8733.619,E2 -8733.619} C_VEL
LIN {X 0,Y 445.55,Z 853.886,A -85,B 0,C 180,E1 -8734.978,E2 -8734.978} C_VEL
LIN {X 0,Y 445.628,Z 849.27,A -85,B 0,C 180,E1 -8736.497,E2 -8736.497} C_VEL
LIN {X 0,Y 445.848,Z 842.563,A -85,B 0,C 180,E1 -8738.157,E2 -8738.157} C_VEL
LIN {X 0,Y 446.127,Z 835.445,A -85,B 0,C 180,E1 -8739.522,E2 -8739.522} C_VEL
LIN {X 0,Y 446.528,Z 826.563,A -85,B 0,C 180,E1 -8740.887,E2 -8740.887} C_VEL
LIN {X 0,Y 447.055,Z 817.422,A -85,B 0,C 180,E1 -8742.023,E2 -8742.023} C_VEL
LIN {X 0,Y 447.591,Z 806.549,A -85,B 0,C 180,E1 -8743.105,E2 -8743.105} C_VEL
LIN {X 0,Y 448.127,Z 795.864,A -85,B 0,C 180,E1 -8743.954,E2 -8743.954} C_VEL
LIN {X 0,Y 448.674,Z 784.008,A -85,B 0,C 180,E1 -8744.689,E2 -8744.689} C_VEL
LIN {X 0,Y 449.109,Z 770.798,A -85,B 0,C 180,E1 -8745.283,E2 -8745.283} C_VEL
LIN {X 0,Y 449.517,Z 757.567,A -85,B 0,C 180,E1 -8745.676,E2 -8745.676} C_VEL
LIN {X 0,Y 450.426,Z 667.43,A -85,B 0,C 180,E1 -8747.227,E2 -8747.227} C_VEL
LIN {X 0,Y 447.225,Z 640.234,A -85,B 0,C 180,E1 -8747.852,E2 -8747.852} C_VEL
LIN {X 0,Y 448.041,Z 620.391,A -85,B 0,C 180,E1 -8750.908,E2 -8750.908} C_VEL
LIN {X 0,Y 448.911,Z 601.998,A -85,B 0,C 180,E1 -8753.775,E2 -8753.775} C_VEL
LIN {X 0,Y 450.066,Z 580.148,A -85,B 0,C 180,E1 -8757.216,E2 -8757.216} C_VEL
LIN {X 0,Y 450.861,Z 565.987,A -85,B 0,C 180,E1 -8759.483,E2 -8759.483} C_VEL
LIN {X 0,Y 449.5,Z 558.341,A -85,B 0,C 180,E1 -8760.819,E2 -8760.819} C_VEL
LIN {X 0,Y 446.466,Z 544.874,A -85,B 0,C 180,E1 -8763.297,E2 -8763.297} C_VEL
LIN {X 0,Y 446.404,Z 544.881,A -85,B 0,C 180,E1 -8766.745,E2 -8766.745} C_VEL
LIN {X 0,Y 446.471,Z 544.87,A -85,B 0,C 180,E1 -8769.527,E2 -8769.527} C_VEL
LIN {X 0,Y 446.432,Z 544.875,A -85,B 0,C 180,E1 -8772.605,E2 -8772.605} C_VEL
LIN {X 0,Y 446.458,Z 544.871,A -85,B 0,C 180,E1 -8775.103,E2 -8775.103} C_VEL
LIN {X 0,Y 446.431,Z 544.868,A -85,B 0,C 180,E1 -8778.609,E2 -8778.609} C_VEL
LIN {X 0,Y 446.447,Z 544.875,A -85,B 0,C 180,E1 -8780.973,E2 -8780.973} C_VEL
LIN {X 0,Y 446.422,Z 544.869,A -85,B 0,C 180,E1 -8784.374,E2 -8784.374} C_VEL
LIN {X 0,Y 446.423,Z 544.87,A -85,B 0,C 180,E1 -8787.638,E2 -8787.638} C_VEL
LIN {X 0,Y 446.449,Z 544.868,A -85,B 0,C 180,E1 -8790.791,E2 -8790.791} C_VEL
LIN {X 0,Y 446.478,Z 544.862,A -85,B 0,C 180,E1 -8793.848,E2 -8793.848} C_VEL
LIN {X 0,Y 446.429,Z 544.868,A -85,B 0,C 180,E1 -8796.823,E2 -8796.823} C_VEL
LIN {X 0,Y 446.444,Z 544.871,A -85,B 0,C 180,E1 -8799.737,E2 -8799.737} C_VEL
LIN {X 0,Y 446.463,Z 544.856,A -85,B 0,C 180,E1 -8802.597,E2 -8802.597} C_VEL
LIN {X 0,Y 446.472,Z 544.872,A -85,B 0,C 180,E1 -8805.412,E2 -8805.412} C_VEL
LIN {X 0,Y 446.517,Z 544.854,A -85,B 0,C 180,E1 -8808.193,E2 -8808.193} C_VEL
LIN {X 0,Y 446.6,Z 544.854,A -85,B 0,C 180,E1 -8811.858,E2 -8811.858} C_VEL
LIN {X 0,Y 446.646,Z 544.844,A -85,B 0,C 180,E1 -8814.583,E2 -8814.583} C_VEL
LIN {X 0,Y 446.664,Z 544.838,A -85,B 0,C 180,E1 -8818.197,E2 -8818.197} C_VEL
LIN {X 0,Y 446.792,Z 544.831,A -85,B 0,C 180,E1 -8820,E2 -8820} C_VEL
LIN {X 0,Y 446.692,Z 544.837,A -85,B 0,C 180,E1 -8822.705,E2 -8822.705} C_VEL
LIN {X 0,Y 446.646,Z 544.842,A -85,B 0,C 180,E1 -8826.324,E2 -8826.324} C_VEL
LIN {X 0,Y 446.538,Z 544.859,A -85,B 0,C 180,E1 -8829.055,E2 -8829.055} C_VEL
LIN {X 0,Y 446.522,Z 544.85,A -85,B 0,C 180,E1 -8832.73,E2 -8832.73} C_VEL
LIN {X 0,Y 446.496,Z 544.866,A -85,B 0,C 180,E1 -8836.228,E2 -8836.228} C_VEL
LIN {X 0,Y 446.47,Z 544.858,A -85,B 0,C 180,E1 -8839.303,E2 -8839.303} C_VEL
LIN {X 0,Y 446.419,Z 544.878,A -85,B 0,C 180,E1 -8842.2,E2 -8842.2} C_VEL
LIN {X 0,Y 446.458,Z 544.861,A -85,B 0,C 180,E1 -8845.152,E2 -8845.152} C_VEL
LIN {X 0,Y 446.486,Z 544.871,A -85,B 0,C 180,E1 -8848.179,E2 -8848.179} C_VEL
LIN {X 0,Y 446.419,Z 544.872,A -85,B 0,C 180,E1 -8851.775,E2 -8851.775} C_VEL
LIN {X 0,Y 446.43,Z 544.872,A -85,B 0,C 180,E1 -8854.523,E2 -8854.523} C_VEL
LIN {X 0,Y 446.417,Z 544.883,A -85,B 0,C 180,E1 -8858.079,E2 -8858.079} C_VEL
LIN {X 0,Y 446.429,Z 544.875,A -85,B 0,C 180,E1 -8860.918,E2 -8860.918} C_VEL
LIN {X 0,Y 446.402,Z 544.875,A -85,B 0,C 180,E1 -8863.846,E2 -8863.846} C_VEL
LIN {X 0,Y 446.399,Z 544.87,A -85,B 0,C 180,E1 -8866.404,E2 -8866.404} C_VEL
LIN {X 0,Y 446.454,Z 544.873,A -85,B 0,C 180,E1 -8869.803,E2 -8869.803} C_VEL
LIN {X 0,Y 446.412,Z 544.871,A -85,B 0,C 180,E1 -8872.121,E2 -8872.121} C_VEL
LIN {X 0,Y 446.433,Z 544.875,A -85,B 0,C 180,E1 -8875.477,E2 -8875.477} C_VEL
LIN {X 0,Y 446.42,Z 544.882,A -85,B 0,C 180,E1 -8878.7,E2 -8878.7} C_VEL
LIN {X 0,Y 446.48,Z 545.009,A -85,B 0,C 180,E1 -8880.635,E2 -8880.635} C_VEL
LIN {X 0,Y 450.243,Z 561.4,A -85,B 0,C 180,E1 -8883.335,E2 -8883.335} C_VEL
